// TwinCAT 3 PLC project UlyssesToolBox
// Title: UlyssesToolBox
// Company: NoCompany
// ProjectVersion: 1.0.0.1
// ProgramVersion: 3.1.4024.0
// project tree:
//   TF04Controller/TempController/ EasyTemp.TcPOU, E_EasyTempState.TcDUT, E_TuneMode.TcDUT, FB_TempSimu.TcPOU, ST_EasyTempPara.TcDUT
//   TF05Motion/SimpleAxis/ E_MoveMode.TcDUT, E_SimpleAxisState.TcDUT, FB_SimpleAxis.TcPOU, ST_AxisSettings.TcDUT
//   TF06Connectivity/TCPIP/ FB_TcpSendReceive.TcPOU, FB_TcpSendReceiving.TcPOU, FB_TcpSendReceivingQueue.TcPOU
//   TF06Connectivity/TCPIP/SimpleClient/ SimpleTcpClient.TcPOU, stConnState.TcDUT, stSktPara.TcDUT
//   TF06Connectivity/TCPIP/TcpTaskQueue2/ FB_SimpleTcpTaskQueue2.TcPOU, ST_TcpTask2.TcDUT, ST_TcpTaskBuffer2.TcDUT
//   TF06Connectivity/TCPIP/TcpTaskQueue/ FB_SimpleTcpTaskQueue.TcPOU, ST_TcpTask.TcDUT, ST_TcpTaskBuffer.TcDUT
//   TF06Connectivity/TCPIP/[obsolete]/ FB_TcpSendReceivingHistroy.TcPOU
//   TF11PlcSystem/AnalogScale/ AnalogScale.TcPOU, AnalogScaleWithAlarm.TcPOU
//   TF11PlcSystem/ET_DoubleBuffer/ DataFileLogger.TcPOU, DoubleBuffer.TcPOU, HRESULT_TO_ADSERROR.TcPOU
//   TF11PlcSystem/File/ FB_FileHandler.TcPOU
//   TF11PlcSystem/IO/ DI_Button.TcPOU, DI_Input.TcPOU, Input.TcPOU, Output.TcPOU
//   TF11PlcSystem/Logger/ E_LogFileSplitMode.TcDUT, ULogger.TcPOU
//   TF11PlcSystem/System/File/ FB_File.TcPOU
//   TF11PlcSystem/System/Pendulum4Tc/ Constants.TcPOU, Day.TcPOU, GVLPendulum.TcGVL, Pendulum4Tc.TcPOU, PtDateTime.TcPOU, PtHelper.TcPOU, PtInterval.TcPOU, PtTimeSource.TcPOU
//   TF11PlcSystem/System/Pendulum4Tc/DUTs/ E_TimeSource.TcDUT, PtWeekDay.TcTLEO, ST_WinsowsTimeZone.TcDUT
//   TF11PlcSystem/System/Pendulum4Tc/Functions/ F_TzInfoBiasToTzStr.TcPOU
//   TF11PlcSystem/System/Pendulum4Tc/Helper/ calcDayNumber.TcPOU, calcPreciseDiff.TcPOU, isDateTimeEqual.TcPOU, isLeapYear.TcPOU, PtPreciseDiff.TcPOU
//   TF11PlcSystem/System/Pendulum4Tc/Interface/ I_PtDateTime.TcIO, I_PtInterval.TcIO, I_PtTimesource.TcIO
//   TF11PlcSystem/System/SystemInfo/ System_AppInfo.TcPOU, System_IpcInfo.TcPOU, System_TaskInfo.TcPOU
//   TF11PlcSystem/System/ SystemPulses.TcPOU
//   TF11PlcSystem/System/Time/DataTypes/ ST_TimeConvertor.TcDUT
//   TF11PlcSystem/System/Time/FunctionBlocks/ FB_TimeConvertorM.TcPOU, FB_Time_Task.TcPOU, Pulse.TcPOU, TimeConvertor.TcPOU
//   TF11PlcSystem/System/Time/Functions/ F_FormatTime.TcPOU, F_SYSTEMTIME_TO_String6.TcPOU
//   TF11PlcSystem/System/Time/[obsolete]/ Base_SysTime.TcPOU, FB_TimeConvertor0.TcPOU, F_TimeStamp13_TO_SYSTEMTIME.TcPOU, PulseWrong.TcPOU
// (motion and I/O tree: see PLC project plc851)
// real-time tasks:
//   TASK PlcTask: cycle T#10ms, priority 20, ADS port 350

// ---- TF04Controller/TempController/E_EasyTempState.TcDUT
{attribute 'qualified_only'}
{attribute 'strict'}
TYPE E_EasyTempState :
(
	Stopped := 0,
	Running := 1,
	Tuning := 2,
	Resetting := 99
);
END_TYPE

// ---- TF04Controller/TempController/E_TuneMode.TcDUT
{attribute 'qualified_only'}
{attribute 'strict'}
TYPE E_TuneMode :
(
	Normal := 0,
	Fast := 1,
	Slow :=2
);
END_TYPE

// ---- TF04Controller/TempController/ST_EasyTempPara.TcDUT
TYPE ST_EasyTempPara :
STRUCT
	bTuned : BOOL;
	stPID : ST_CTRL_ParaController;
	stPara: ST_CTRL_TempCtrlParameter;
END_STRUCT
END_TYPE

// ---- TF05Motion/SimpleAxis/E_MoveMode.TcDUT
{attribute 'qualified_only'}
{attribute 'strict'}
TYPE E_MoveMode :
(
	NotMove := 0,
	MoveAbs := 1,
	MoveMod := 2,
	MoveRel := 3

);
END_TYPE

// ---- TF05Motion/SimpleAxis/E_SimpleAxisState.TcDUT
{attribute 'qualified_only'}
{attribute 'strict'}
TYPE E_SimpleAxisState :
(
	Waiting := 0,
	BeforeJog := 10,
	Joging :=11,
	JogDone := 18,
	
	BeforeMovePos :=20,
	MovingAbs := 21,
	MovingMod :=23,
	MovingRel := 24,
	MovePosDone := 28,
	
	BeforeMoveVelo := 30,
	MovingVelo := 31,
	MoveVeloStop := 32,
	MoveVeloDone := 38,
	
	
	BeforeHoming := 50,
	Homing :=51,
	FinishHoming := 52,
	HomeToZero := 53,
	HomeDone :=58,

	Aborted := 90,
	Error :=99

);
END_TYPE

// ---- TF05Motion/SimpleAxis/ST_AxisSettings.TcDUT
TYPE ST_AxisSettings :
STRUCT
	MovePosAcc : LREAL;
	MovePosDec : LREAL;
	MovePosJerk : LREAL;
	
	MoveVeloAcc : LREAL;
	MoveVeloDec : LREAL;
	MoveVeloJerk : LREAL;
	MoveVeloDirection : MC_Direction := MC_Positive_Direction;
	
	JogAcc : LREAL;
	JogDec : LREAL;
	JogJerk : LREAL;
	
	HomeVelo : LREAL := 10;
	HomeAcc : LREAL;
	HomeDec : LREAL;
	HomeJerk : LREAL;
	HomeSetpos : LREAL := 0;
	HomeSignal : BOOL;
	HomePosLimit : BOOL;
	HomeNegLimit : BOOL;
END_STRUCT
END_TYPE

// ---- TF06Connectivity/TCPIP/SimpleClient/stConnState.TcDUT
TYPE stConnState :
STRUCT
	bConnected : BOOL;
	hSocket : T_HSOCKET;
	eState : E_SocketConnectionState;
	bError : BOOL;
	nErrId : UDINT;
END_STRUCT
END_TYPE

// ---- TF06Connectivity/TCPIP/SimpleClient/stSktPara.TcDUT
TYPE stSktPara :
STRUCT
	AutoReconnect : BOOL;
	EnableSendLog : BOOL;
	EnableRecvLog : BOOL;
	SendRecvTimeOut : TIME := T#3S;
	
END_STRUCT
END_TYPE

// ---- TF06Connectivity/TCPIP/TcpTaskQueue2/ST_TcpTask2.TcDUT
{attribute 'pack_mode' := '1'}
TYPE ST_TcpTask2 :
STRUCT
	TaskName : STRING(24);
	TaskType : INT; (* 0:Once, 1:Regular *)
	pData : PVOID;
	nData : UDINT;
END_STRUCT
END_TYPE

// ---- TF06Connectivity/TCPIP/TcpTaskQueue2/ST_TcpTaskBuffer2.TcDUT
{attribute 'pack_mode' := '1'}
TYPE ST_TcpTaskBuffer2 :
STRUCT
	BufferInfo : UDINT;
	TaskData : ST_TcpTask2;
END_STRUCT
END_TYPE

// ---- TF06Connectivity/TCPIP/TcpTaskQueue/ST_TcpTask.TcDUT
{attribute 'pack_mode' := '1'}
TYPE ST_TcpTask :
STRUCT
	TaskName : STRING(24);
	TaskType : INT; (* 0:Once, 1:Regular *)
	TaskData : ARRAY[0..255] OF BYTE;
END_STRUCT
END_TYPE

// ---- TF06Connectivity/TCPIP/TcpTaskQueue/ST_TcpTaskBuffer.TcDUT
{attribute 'pack_mode' := '1'}
TYPE ST_TcpTaskBuffer :
STRUCT
	BufferInfo : ARRAY[0..3] OF BYTE;
	TaskData : ST_TcpTask;
END_STRUCT
END_TYPE

// ---- TF11PlcSystem/Logger/E_LogFileSplitMode.TcDUT
{attribute 'qualified_only'}
{attribute 'strict'}
TYPE E_LogFileSplitMode :
(
	eDontSplit := 0,
	eSplitByDay := 1,
	eSplitByHour := 2
);
END_TYPE

// ---- TF11PlcSystem/System/Pendulum4Tc/DUTs/E_TimeSource.TcDUT
{attribute 'qualified_only'}
{attribute 'strict'}
TYPE E_TimeSource :
(
	FileTime := 0,
	DcTaskInfo := 1,
	fbLocalSystemTime := 2
);
END_TYPE

// ---- TF11PlcSystem/System/Pendulum4Tc/DUTs/PtWeekDay.TcTLEO
{attribute 'qualified_only'}
{attribute 'strict'}
TYPE PtWeekDay :
(
	MONDAY := 0,
    TUESDAY := 1,
    WEDNESDAY := 2,
    THURSDAY := 3,
    FRIDAY := 4,
    SATURDAY := 5,
    SUNDAY := 6
);
END_TYPE

// ---- TF11PlcSystem/System/Pendulum4Tc/DUTs/ST_WinsowsTimeZone.TcDUT
TYPE ST_WinsowsTimeZone :
STRUCT
	AUS_Central_Standard_Time	: STRING	:=	 'Australia/Darwin';
	AUS_Eastern_Standard_Time	: STRING	:=	 'Australia/Sydney';
	Afghanistan_Standard_Time	: STRING	:=	 'Asia/Kabul';
	Alaskan_Standard_Time	: STRING	:=	 'America/Anchorage';
	Aleutian_Standard_Time	: STRING	:=	 'America/Adak';
	Altai_Standard_Time	: STRING	:=	 'Asia/Barnaul';
	Arab_Standard_Time	: STRING	:=	 'Asia/Riyadh';
	Arabian_Standard_Time	: STRING	:=	 'Asia/Dubai';
	Arabic_Standard_Time	: STRING	:=	 'Asia/Baghdad';
	Argentina_Standard_Time	: STRING	:=	 'America/Buenos_Aires';
	Astrakhan_Standard_Time	: STRING	:=	 'Europe/Astrakhan';
	Atlantic_Standard_Time	: STRING	:=	 'America/Halifax';
	Aus_Central_Wdot_Standard_Time	: STRING	:=	 'Australia/Eucla';
	Azerbaijan_Standard_Time	: STRING	:=	 'Asia/Baku';
	Azores_Standard_Time	: STRING	:=	 'Atlantic/Azores';
	Bahia_Standard_Time	: STRING	:=	 'America/Bahia';
	Bangladesh_Standard_Time	: STRING	:=	 'Asia/Dhaka';
	Belarus_Standard_Time	: STRING	:=	 'Europe/Minsk';
	Bougainville_Standard_Time	: STRING	:=	 'Pacific/Bougainville';
	Canada_Central_Standard_Time	: STRING	:=	 'America/Regina';
	Cape_Verde_Standard_Time	: STRING	:=	 'Atlantic/Cape_Verde';
	Caucasus_Standard_Time	: STRING	:=	 'Asia/Yerevan';
	Cendot_Australia_Standard_Time	: STRING	:=	 'Australia/Adelaide';
	Central_America_Standard_Time	: STRING	:=	 'America/Guatemala';
	Central_Asia_Standard_Time	: STRING	:=	 'Asia/Almaty';
	Central_Brazilian_Standard_Time	: STRING	:=	 'America/Cuiaba';
	Central_Europe_Standard_Time	: STRING	:=	 'Europe/Budapest';
	Central_European_Standard_Time	: STRING	:=	 'Europe/Warsaw';
	Central_Pacific_Standard_Time	: STRING	:=	 'Pacific/Guadalcanal';
	Central_Standard_Time	: STRING	:=	 'America/Chicago';
	Central_Standard_Time_Mexico	: STRING	:=	 'America/Mexico_City';
	Chatham_Islands_Standard_Time	: STRING	:=	 'Pacific/Chatham';
	China_Standard_Time	: STRING	:=	 'Asia/Shanghai';
	Cuba_Standard_Time	: STRING	:=	 'America/Havana';
	Dateline_Standard_Time	: STRING	:=	 'Etc/GMT+12';
	Edot_Africa_Standard_Time	: STRING	:=	 'Africa/Nairobi';
	Edot_Australia_Standard_Time	: STRING	:=	 'Australia/Brisbane';
	Edot_Europe_Standard_Time	: STRING	:=	 'Europe/Chisinau';
	Edot_South_America_Standard_Time	: STRING	:=	 'America/Sao_Paulo';
	Easter_Island_Standard_Time	: STRING	:=	 'Pacific/Easter';
	Eastern_Standard_Time	: STRING	:=	 'America/New_York';
	Eastern_Standard_Time_Mexico	: STRING	:=	 'America/Cancun';
	Egypt_Standard_Time	: STRING	:=	 'Africa/Cairo';
	Ekaterinburg_Standard_Time	: STRING	:=	 'Asia/Yekaterinburg';
	FLE_Standard_Time	: STRING	:=	 'Europe/Kiev';
	Fiji_Standard_Time	: STRING	:=	 'Pacific/Fiji';
	GMT_Standard_Time	: STRING	:=	 'Europe/London';
	GTB_Standard_Time	: STRING	:=	 'Europe/Bucharest';
	Georgian_Standard_Time	: STRING	:=	 'Asia/Tbilisi';
	Greenland_Standard_Time	: STRING	:=	 'America/Godthab';
	Greenwich_Standard_Time	: STRING	:=	 'Atlantic/Reykjavik';
	Haiti_Standard_Time	: STRING	:=	 'America/Port-au-Prince';
	Hawaiian_Standard_Time	: STRING	:=	 'Pacific/Honolulu';
	India_Standard_Time	: STRING	:=	 'Asia/Calcutta';
	Iran_Standard_Time	: STRING	:=	 'Asia/Tehran';
	Israel_Standard_Time	: STRING	:=	 'Asia/Jerusalem';
	Jordan_Standard_Time	: STRING	:=	 'Asia/Amman';
	Kaliningrad_Standard_Time	: STRING	:=	 'Europe/Kaliningrad';
	Korea_Standard_Time	: STRING	:=	 'Asia/Seoul';
	Libya_Standard_Time	: STRING	:=	 'Africa/Tripoli';
	Line_Islands_Standard_Time	: STRING	:=	 'Pacific/Kiritimati';
	Lord_Howe_Standard_Time	: STRING	:=	 'Australia/Lord_Howe';
	Magadan_Standard_Time	: STRING	:=	 'Asia/Magadan';
	Magallanes_Standard_Time	: STRING	:=	 'America/Punta_Arenas';
	Marquesas_Standard_Time	: STRING	:=	 'Pacific/Marquesas';
	Mauritius_Standard_Time	: STRING	:=	 'Indian/Mauritius';
	Middle_East_Standard_Time	: STRING	:=	 'Asia/Beirut';
	Montevideo_Standard_Time	: STRING	:=	 'America/Montevideo';
	Morocco_Standard_Time	: STRING	:=	 'Africa/Casablanca';
	Mountain_Standard_Time	: STRING	:=	 'America/Denver';
	Mountain_Standard_Time_Mexico	: STRING	:=	 'America/Chihuahua';
	Myanmar_Standard_Time	: STRING	:=	 'Asia/Rangoon';
	Ndot_Central_Asia_Standard_Time	: STRING	:=	 'Asia/Novosibirsk';
	Namibia_Standard_Time	: STRING	:=	 'Africa/Windhoek';
	Nepal_Standard_Time	: STRING	:=	 'Asia/Katmandu';
	New_Zealand_Standard_Time	: STRING	:=	 'Pacific/Auckland';
	Newfoundland_Standard_Time	: STRING	:=	 'America/St_Johns';
	Norfolk_Standard_Time	: STRING	:=	 'Pacific/Norfolk';
	North_Asia_East_Standard_Time	: STRING	:=	 'Asia/Irkutsk';
	North_Asia_Standard_Time	: STRING	:=	 'Asia/Krasnoyarsk';
	North_Korea_Standard_Time	: STRING	:=	 'Asia/Pyongyang';
	Omsk_Standard_Time	: STRING	:=	 'Asia/Omsk';
	Pacific_SA_Standard_Time	: STRING	:=	 'America/Santiago';
	Pacific_Standard_Time	: STRING	:=	 'America/Los_Angeles';
	Pacific_Standard_Time_Mexico	: STRING	:=	 'America/Tijuana';
	Pakistan_Standard_Time	: STRING	:=	 'Asia/Karachi';
	Paraguay_Standard_Time	: STRING	:=	 'America/Asuncion';
	Romance_Standard_Time	: STRING	:=	 'Europe/Paris';
	Russia_Time_Zone_10	: STRING	:=	 'Asia/Srednekolymsk';
	Russia_Time_Zone_11	: STRING	:=	 'Asia/Kamchatka';
	Russia_Time_Zone_3	: STRING	:=	 'Europe/Samara';
	Russian_Standard_Time	: STRING	:=	 'Europe/Moscow';
	SA_Eastern_Standard_Time	: STRING	:=	 'America/Cayenne';
	SA_Pacific_Standard_Time	: STRING	:=	 'America/Bogota';
	SA_Western_Standard_Time	: STRING	:=	 'America/La_Paz';
	SE_Asia_Standard_Time	: STRING	:=	 'Asia/Bangkok';
	Saint_Pierre_Standard_Time	: STRING	:=	 'America/Miquelon';
	Sakhalin_Standard_Time	: STRING	:=	 'Asia/Sakhalin';
	Samoa_Standard_Time	: STRING	:=	 'Pacific/Apia';
	Sao_Tome_Standard_Time	: STRING	:=	 'Africa/Sao_Tome';
	Saratov_Standard_Time	: STRING	:=	 'Europe/Saratov';
	Singapore_Standard_Time	: STRING	:=	 'Asia/Singapore';
	South_Africa_Standard_Time	: STRING	:=	 'Africa/Johannesburg';
	Sri_Lanka_Standard_Time	: STRING	:=	 'Asia/Colombo';
	Sudan_Standard_Time	: STRING	:=	 'Africa/Khartoum';
	Syria_Standard_Time	: STRING	:=	 'Asia/Damascus';
	Taipei_Standard_Time	: STRING	:=	 'Asia/Taipei';
	Tasmania_Standard_Time	: STRING	:=	 'Australia/Hobart';
	Tocantins_Standard_Time	: STRING	:=	 'America/Araguaina';
	Tokyo_Standard_Time	: STRING	:=	 'Asia/Tokyo';
	Tomsk_Standard_Time	: STRING	:=	 'Asia/Tomsk';
	Tonga_Standard_Time	: STRING	:=	 'Pacific/Tongatapu';
	Transbaikal_Standard_Time	: STRING	:=	 'Asia/Chita';
	Turkey_Standard_Time	: STRING	:=	 'Europe/Istanbul';
	Turks_And_Caicos_Standard_Time	: STRING	:=	 'America/Grand_Turk';
	US_Eastern_Standard_Time	: STRING	:=	 'America/Indianapolis';
	US_Mountain_Standard_Time	: STRING	:=	 'America/Phoenix';
	UTC	: STRING	:=	 'Etc/GMT';
	UTCplus12	: STRING	:=	 'Etc/GMT-12';
	UTCplus13	: STRING	:=	 'Etc/GMT-13';
	UTCminus02	: STRING	:=	 'Etc/GMT+2';
	UTCminus08	: STRING	:=	 'Etc/GMT+8';
	UTCminus09	: STRING	:=	 'Etc/GMT+9';
	UTCminus11	: STRING	:=	 'Etc/GMT+11';
	Ulaanbaatar_Standard_Time	: STRING	:=	 'Asia/Ulaanbaatar';
	Venezuela_Standard_Time	: STRING	:=	 'America/Caracas';
	Vladivostok_Standard_Time	: STRING	:=	 'Asia/Vladivostok';
	Wdot_Australia_Standard_Time	: STRING	:=	 'Australia/Perth';
	Wdot_Central_Africa_Standard_Time	: STRING	:=	 'Africa/Lagos';
	Wdot_Europe_Standard_Time	: STRING	:=	 'Europe/Berlin';
	Wdot_Mongolia_Standard_Time	: STRING	:=	 'Asia/Hovd';
	West_Asia_Standard_Time	: STRING	:=	 'Asia/Tashkent';
	West_Bank_Standard_Time	: STRING	:=	 'Asia/Hebron';
	West_Pacific_Standard_Time	: STRING	:=	 'Pacific/Port_Moresby';
	Yakutsk_Standard_Time	: STRING	:=	 'Asia/Yakutsk';

END_STRUCT
END_TYPE

// ---- TF11PlcSystem/System/Time/DataTypes/ST_TimeConvertor.TcDUT
TYPE ST_TimeConvertor :
STRUCT
		(* #########################  System  ######################### *)
		
	(* Alias: -- *)
	(* Size: 32-bit *)
	(* Range: 0=>1970-01-01 2^32-1=>2106-02-07 *)
	(* Resolution: 1s, only the day is displayed *)
	(* https://infosys.beckhoff.com/english.php?content=../content/1033/tc3_plc_intro/2529415819.html&id=7132877304198979715 *)
	(* Native *)
	Date_D : DATE;
	
	(* Alias: -- *)
	(* Size: 32-bit *)
	(* Range: 0=>00:00:00.000 86399999=>23:59:59.999 *)
	(* Resolution: 1ms *)
	(* https://infosys.beckhoff.com/english.php?content=../content/1033/tc3_plc_intro/2529415819.html&id=7132877304198979715 *)
	(* Native *)
	TimeOfDay_TOD : TIME_OF_DAY;
	
	(* Alias: -- *)
	(* Size: 32-bit *)
	(* Range: 0=>1970-01-01 00:00:00 2^32-1=>2106-02-07 06:28:15 *)
	(* Resolution: 1s *)
	(* https://infosys.beckhoff.com/english.php?content=../content/1033/tc3_plc_intro/2529415819.html&id=7132877304198979715 *)
	(* Native *)
	DateAndTime_DT : DATE_AND_TIME;
	
	(* Alias: -- *)
	(* Size: 64-bit *)
	(* Range: 0=>1970-01-01 2^64-1=>2554-07-21 *)
	(* Resolution: 1ns *)
	(* https://infosys.beckhoff.com/english.php?content=../content/1033/tc3_plc_intro/2529415819.html&id=7132877304198979715 *)
	(* Only For >=4026.0 *)
	//LDate_LDT : LDATE;
	
	(* Alias: -- *)
	(* Size: 64-bit *)
	(* Range: 0=>00:00:00.000000000 2^64-1=>23:59:59.999999999 *)
	(* Resolution: 1ns *)
	(* https://infosys.beckhoff.com/english.php?content=../content/1033/tc3_plc_intro/2529415819.html&id=7132877304198979715 *)
	(* Only For >=4026.0 *)
	//LTimeOfDay_LTOD : LTIME_OF_DAY;
	
	(* Alias: -- *)
	(* Size: 64-bit *)
	(* Range: 0=>1970-01-01 00:00:00.000000000 2^64-1=>2554-07-21 23:34:33.709551615 *)
	(* Resolution: 1ns *)
	(* https://infosys.beckhoff.com/english.php?content=../content/1033/tc3_plc_intro/2529415819.html&id=7132877304198979715 *)
	(* Only For >=4026.0 *)
	//LDateAndTime_LDT : LDATE_AND_TIME;
	
		(* #########################  Tc2_Utilities  ######################### *)
	
	(* Alias: T_ULARGE_INTEGER -> Struct of 2 DWORD *)
	(* Size: 64-bit *)
	(* Range: -- *)
	(* Resolution: 100ns *)
	(* obsolete! *)
	FileTime : T_FILETIME;
	
	(* Alias: ULINT *)
	(* Size: 64-bit *)
	(* Range: 0=>1601-01-01 00:00:00.0000000 2^64-1=>2185-11-09 23:34:33.9999999 *)
	(* Resolution: 100ns *)
	(* https://infosys.beckhoff.com/english.php?content=../content/1033/tcplclib_tc2_utilities/10462547339.html&id= *)
	(* Recommend! *)
	FileTime64 : T_FILETIME64;
	
	(* Alias: Struct of 8 WORD *)
	(* Size: 128-bit *)
	(* Range: 1970-01-01 Sunday 00:00:00.000  2106-12-31 Saturday 23:59:59.999 *)
	(* Resolution: 1ms *)
	(* https://infosys.beckhoff.com/english.php?content=../content/1033/tcplclib_tc2_utilities/35393035.html&id=8702657298802174446 *)
	(* Recommend! *)
	TimeStruct : TIMESTRUCT;
	
	(* Alias: Struct of 6 WORD *)
	(* Size: 96-bit *)
	(* Range: Week0 Day0 00:00:00.000  Week65535 Day7 23:59:59.999 *)
	(* Resolution: 1ms *)
	(* https://infosys.beckhoff.com/english.php?content=../content/1033/tcplclib_tc2_utilities/35353099.html&id=8265378500365774535 *)
	(* What's this??  weeks + days *)
	(* NOT Recommend! *)
	OtStruct : OTSTRUCT;
	
		(* #########################  Tc2_EtherCAT  ######################### *)
		
	(* Alias: T_ULARGE_INTEGER -> Struct of 2 DWORD *)
	(* Size: 64-bit *)
	(* Range: -- *)
	(* Resolution: 1ns *)
	(* obsolete! *)
	DcTime : T_DCTIME;
	
	(* Alias: UDINT *)
	(* Size: 32-bit *)
	(* Range: +-2147s *)
	(* Resolution: 1ns *)
	(* NOT Recommend! *)
	DcTime32 : T_DCTIME32; 
	
	(* Alias: ULINT *)
	(* Size: 64-bit *)
	(* Range: 0=>2000-01-01 00:00:00.000000000 2^64-1=>2584-11-09 23:34:33.999999999 *)
	(* Resolution: 1ns *)
	(* Recommend! *)
	DcTime64 : T_DCTIME64;

		(* #########################  Custom & Others  ######################### *)
	
	Unix : UDINT;
	UnixEx : ULINT;
	//Unix64
END_STRUCT
END_TYPE

// ---- TF11PlcSystem/System/Pendulum4Tc/GVLPendulum.TcGVL
//{attribute 'qualified_only'}
VAR_GLOBAL
	Pendulum : Pendulum4Tc;
END_VAR

// ---- TF11PlcSystem/System/Pendulum4Tc/Interface/I_PtDateTime.TcIO
INTERFACE I_PtDateTime

END_INTERFACE

// ---- TF11PlcSystem/System/Pendulum4Tc/Interface/I_PtInterval.TcIO
INTERFACE I_PtInterval

METHOD inMonth : DINT
VAR_INPUT
END_VAR
END_METHOD

METHOD inYears : DINT
VAR_INPUT
END_VAR
END_METHOD

END_INTERFACE

// ---- TF11PlcSystem/System/Pendulum4Tc/Interface/I_PtTimesource.TcIO
INTERFACE I_PtTimesource

METHOD getDateTime : PtDateTime
VAR_INPUT
END_VAR
END_METHOD

END_INTERFACE

// ---- TF11PlcSystem/System/Pendulum4Tc/Pendulum4Tc.TcPOU
FUNCTION_BLOCK Pendulum4Tc
VAR_INPUT
	TimeSourceDateTime : I_PtTimesource;
END_VAR
VAR_OUTPUT
END_VAR
VAR
	_DateTime : PtDateTime;
	_Interval : PtInterval;
END_VAR


_DateTime := TimeSourceDateTime.getDateTime();

METHOD New : PtDateTime
VAR_INPUT
	Year : DINT;
	Month : DINT;
	Day : DINT;
	Hour : DINT;
	Minute : DINT;
	Second : DINT;
	Microsecond : DINT;
	TimeZone : DINT;
END_VAR
New.Set(
	Year:= Year, 
	Month:= Month, 
	Day:= Day, 
	Hour:= Hour, 
	Minute:= Minute, 
	Second:= Second, 
	Microsecond:= Microsecond, 
	TimeZone:= TimeZone);
END_METHOD

METHOD Now : PtDateTime
VAR_INPUT
END_VAR
Now := _DateTime;
END_METHOD

END_FUNCTION_BLOCK

// ---- TF11PlcSystem/System/Pendulum4Tc/PtDateTime.TcPOU
FUNCTION_BLOCK PtDateTime IMPLEMENTS I_PtDateTime
VAR_INPUT
END_VAR
VAR_OUTPUT
END_VAR
VAR
	_Year : DINT;
	_Month : DINT;
	_Day : DINT;
	_Hour : DINT;
	_Minute : DINT;
	_Second : DINT;
	_Microsecond : DINT;
	_TimeZone : DINT;
	
END_VAR

PROPERTY Day : DINT
GET
Day := _Day;
END_GET
SET
_Day := Day;
END_SET
END_PROPERTY

METHOD Diff : I_PtInterval
VAR_INPUT
	TargetDateTime : PtDateTime;
END_VAR
//Diff.Set(THIS^,TargetDateTime,TRUE);
Pendulum._interval.Set(THIS^,TargetDateTime,TRUE);
Diff := Pendulum._interval;
END_METHOD

PROPERTY Hour : DINT
GET
Hour := _Hour;
END_GET
SET
_Hour := Hour;
END_SET
END_PROPERTY

PROPERTY Microsecond : DINT
GET
Microsecond := _Microsecond;
END_GET
SET
_Microsecond := Microsecond;
END_SET
END_PROPERTY

PROPERTY Minute : DINT
GET
Minute := _Minute;
END_GET
SET
_Minute := Minute;
END_SET
END_PROPERTY

PROPERTY Month : DINT
GET
Month := _Month;
END_GET
SET
_Month := Month;
END_SET
END_PROPERTY

PROPERTY Second : DINT
GET
Second := _Second;
END_GET
SET
_Second := Second;
END_SET
END_PROPERTY

METHOD Set //: PtDateTime
VAR_INPUT
	Year : DINT;
	Month : DINT;
	Day : DINT;
	Hour : DINT;
	Minute : DINT;
	Second : DINT;
	Microsecond : DINT;
	TimeZone : DINT;
END_VAR
THIS^._Year := Year;
THIS^._Month := Month;
THIS^._Day := Day;
THIS^._Hour := Hour;
THIS^._Minute := Minute;
THIS^._Second := Second;
THIS^._Microsecond := Microsecond;
THIS^._TimeZone := TimeZone;
END_METHOD

PROPERTY TimeZone : DINT
GET
TimeZone := _TimeZone;
END_GET
SET
_TimeZone := TimeZone;
END_SET
END_PROPERTY

PROPERTY Year : DINT
GET
Year := _Year;
END_GET
SET
_Year := Year;
END_SET
END_PROPERTY

END_FUNCTION_BLOCK

// ---- TF11PlcSystem/System/Pendulum4Tc/Day.TcPOU
FUNCTION_BLOCK Day
VAR_INPUT
	
END_VAR
VAR_OUTPUT
END_VAR
VAR
END_VAR

END_FUNCTION_BLOCK

// ---- TF11PlcSystem/System/Pendulum4Tc/PtInterval.TcPOU
FUNCTION_BLOCK PtInterval IMPLEMENTS I_PtInterval
VAR_INPUT
END_VAR
VAR_OUTPUT
END_VAR
VAR
	_Start : PtDateTime;
	_End : PtDateTime;
	_Absolute : BOOL;
	
	_DeltaYears : DINT;
	_DeltaMonths : DINT;
	_DeltaDays : DINT;
END_VAR

PROPERTY Absolute : BOOL
GET
Absolute := _Absolute;
END_GET
SET
_Absolute := Absolute;
END_SET
END_PROPERTY

PROPERTY End : PtDateTime
GET
End := _End;
END_GET
SET
_End := End;
END_SET
END_PROPERTY

METHOD inMonth : DINT
VAR_INPUT
END_VAR
inMonth := ABS(_Start.Month - _End.Month);
END_METHOD

METHOD inYears : DINT
VAR_INPUT
END_VAR
inYears := ABS(_Start.Year - _End.Year);
END_METHOD

METHOD Set //: BOOL
VAR_INPUT
	Start : PtDateTime;
	End : PtDateTime;
	Absolute : BOOL;
END_VAR
_Start := Start;
_End := End;
_Absolute := Absolute;

_DeltaYears := ABS(_Start.Year - _End.Year);
_DeltaMonths := ABS(_Start.Month - _End.Month);
_DeltaDays := ABS(_Start.Day - End.Day);
END_METHOD

PROPERTY Start : PtDateTime
GET
END_GET
SET
_Start := Start;
END_SET
END_PROPERTY

END_FUNCTION_BLOCK

// ---- TF04Controller/TempController/EasyTemp.TcPOU
FUNCTION_BLOCK EasyTemp
VAR_INPUT
	bStart : BOOL;
	bTune : BOOL;
	TuneMode : E_TuneMode := E_TuneMode.Normal;
	bReset : BOOL;
	SensorTemp : LREAL;
	TargetTemp : LREAL;
	
END_VAR
VAR_IN_OUT
	EasyTempPara : ST_EasyTempPara;
END_VAR
VAR_OUTPUT
	State : E_EasyTempState;
	fAnalog : LREAL;
	bPWMPos : BOOL;
	bPWMNeg : BOOL;
	bDigPos : BOOL;
	bDigNeg : BOOL;
	fMaxOverShoot: LREAL;
	tStartUpTime: TIME;
	eControlState: Tc2_TempController.E_CTRL_STATE;
	bError: BOOL;
	eErrorId: Tc2_TempController.E_CTRL_ErrorCodes;
	fTempVelo: LREAL;
	
END_VAR
VAR

	rTrigStart : R_TRIG;
	fTrigStart : F_TRIG;
	rTrigTune : R_TRIG;
	rTrigReset : R_TRIG;
	//状态机
	_State : E_EasyTempState;
	rTrigStateReq : R_TRIG;
	fbTemp : FB_CTRL_TempController;


END_VAR

ParaUpdate();


rTrigStart(CLK:= bStart, Q=> );
fTrigStart(CLK:= bStart, Q=> );
rTrigTune(CLK:= bTune, Q=> );
rTrigStateReq(CLK:= rTrigStart.Q XOR fTrigStart.Q XOR rTrigTune.Q, Q=> );
rTrigReset(CLK:= bReset, Q=> );
IF rTrigReset.Q THEN
	_State := E_EasyTempState.Resetting;
END_IF
CASE _State OF
E_EasyTempState.Stopped:
	IF rTrigStateReq.Q THEN
		IF rTrigStart.Q THEN
			IF EasyTempPara.bTuned THEN
				_State := E_EasyTempState.Running;
			END_IF
		ELSIF fTrigStart.Q THEN
			//no action
		ELSIF rTrigTune.Q THEN
			_State := E_EasyTempState.Tuning;
		END_IF
	END_IF
	fbTemp.eCtrlMode := E_CTRL_MODE.eCTRL_MODE_IDLE;
	
E_EasyTempState.Tuning:
	IF rTrigStateReq.Q THEN
		IF rTrigStart.Q THEN
			//no action
		ELSIF fTrigStart.Q THEN
			//no action
		ELSIF rTrigTune.Q THEN
			//no action
		END_IF
	END_IF
	IF fbTemp.eCtrlMode = E_CTRL_MODE.eCTRL_MODE_TUNE AND
		(fbTemp.eCtrlState = E_CTRL_STATE.eCTRL_STATE_TUNED OR fbTemp.bError)THEN
		_State := E_EasyTempState.Stopped;
		IF fbTemp.eCtrlState = E_CTRL_STATE.eCTRL_STATE_TUNED THEN
			EasyTempPara.stPID := fbTemp.sParaControllerInternal;
			EasyTempPara.bTuned := TRUE;
		END_IF
	ELSE
		fbTemp.eCtrlMode := E_CTRL_MODE.eCTRL_MODE_TUNE;
	END_IF
	
E_EasyTempState.Running:
	IF rTrigStateReq.Q THEN
		IF rTrigStart.Q THEN
			//no action
		ELSIF fTrigStart.Q THEN
			_State := E_EasyTempState.Stopped;
		ELSIF rTrigTune.Q THEN
			//no action
		END_IF
	END_IF
	fbTemp.eCtrlMode := E_CTRL_MODE.eCTRL_MODE_ACTIVE;
E_EasyTempState.Resetting:
	fbTemp.eCtrlMode := E_CTRL_MODE.eCTRL_MODE_RESET;
	IF fbTemp.eCtrlState = E_CTRL_STATE.eCTRL_STATE_IDLE THEN
		_State := E_EasyTempState.Stopped;
	END_IF
END_CASE
State := _State;



fbTemp.sParaControllerExternal := EasyTempPara.stPID;
fbTemp.fW1 := TargetTemp;
fbTemp.fX := SensorTemp;
fbTemp(
	eCtrlMode:= , 
	bSelSetpoint:= , 
	fW1:= , 
	fW2:= , 
	fX:= , 
	fYManual:= , 
	bOpenThermocouple:= , 
	bReverseThermocouple:= , 
	bBackVoltage:= , 
	bLeakage:= , 
	bShortCircuit:= , 
	bOpenCircuit:= , 
	sParaControllerExternal:= , 
	sControllerParameter:= EasyTempPara.stPara, 
	fYAnalog=> fAnalog, 
	bYPWMPos=> bPWMPos, 
	bYPWMNeg=> bPWMNeg, 
	bYDigPos=> bDigPos, 
	bYDigNeg=> bDigNeg, 
	dwAlarm=> , 
	fMaxOverShoot=> fMaxOverShoot, 
	tStartUpTime=> tStartUpTime, 
	eCtrlState=> eControlState, 
	sParaControllerInternal=> , 
	bError=> bError, 
	eErrorId=> eErrorId, 
	fYP=> , 
	fYI=> , 
	fYD=> , 
	fTempVelo=> fTempVelo);

METHOD PRIVATE ParaUpdate : BOOL
VAR_INPUT
END_VAR

			(*	常规参数General parameters	*)
(* 控制器操作模式(见下方) *)
(*
eCTRL_ControlMode_HEATING = 1 : 加热
eCTRL_ControlMode_COOLING = 2 : 降温
eCTRL_ControlMode_HEATING_COOLING = 3 : 加热&降温
*)
EasyTempPara.stPara.iMode							:= E_CTRL_ControlMode.eCTRL_ControlMode_HEATING ;
(* 定义发生错误后的行为 *)
(*
eCTRL_ReactionOnFailure_NoFailure : 没有错误
eCTRL_ReactionOnFailure_StopController : 停止
eCTRL_ReactionOnFailure_SetManMode : 设定为手动模式输出
eCTRL_ReactionOnFailure_SetYMax : 设定为最大输出
eCTRL_ReactionOnFailure_SetYMin : 设定为最小输出
eCTRL_ReactionOnFailure_SetYMean : 设定为平均输出
*)
EasyTempPara.stPara.iReactionOnFailure				:= E_CTRL_ReactionOnFailure.eCTRL_ReactionOnFailure_StopController ;
(* TRUE = 外部参数，FALSE = 内部参数 (取决于自整定) *)
EasyTempPara.stPara.bSelCtrlParameterSet			:= TRUE;
(* 报警掩码（见下文）。 *)
(*
Bit0 : 硬件:温度传感器开路,对应bOpenThermocouple引脚
Bit1 : 硬件:温度传感器反接,对应bReverseThermocouple引脚
Bit2 : 硬件:温度传感器电压过高,对应bBackVoltage引脚
Bit4 : 硬件:温度传感器漏电流,对应bLeakage引脚
Bit5 : 硬件:温度传感器短路,对应bShortCircuit引脚
Bit6 : 硬件:温度传感器开路,对应bOpenCircuit引脚
Bit8 : 软件:温度低于L
Bit9 : 软件:温度低于LL
Bit10: 软件:温度高于H
Bit11: 软件:温度高于HH
Bit12: 软件:温度高于AbsoluteHigh
Bit13: 软件:温度低于AbsoluteLow
*)
EasyTempPara.stPara.dwAlarmSupp						:= 16#FF_FF_FF_FF ;
(* 控制器的采样时间。在采样时间的过程中，控制器重新计算控制值。 *)
EasyTempPara.stPara.tCtrlCycleTime					:= T#100MS	 ;
(* 任务周期时间。用这个时间间隔调用FB。 *)
EasyTempPara.stPara.tTaskCycleTime					:= T#10MS ;

			(*	自整定参数Tuning parameters	*)
(* 确定自整定顺序（见下文）。 *)
EasyTempPara.stPara.iTuningMode						:= eCTRL_TuneMode_heating ;
(* 等待时间，直到稳定后再进行自整定。 *)
EasyTempPara.stPara.tTuneStabilisation				:= T#10S;
(* 设定点的百分比值，从该值开始系统切换到闭环控制。 *)
EasyTempPara.stPara.fEndTunePercentHeating			:= 100.0 ;
(* 自整定过程中控制值的阶跃变化。 *)
EasyTempPara.stPara.fYTuneHeating					:= 60.0 ;
(* 加热时切换到自整定时的控制值 *)
EasyTempPara.stPara.fYStableHeating					:= 0 ;
(* 设定点的百分比值，从该值开始系统切换到闭环控制。 *)
EasyTempPara.stPara.fEndTunePercentCooling			:= 20 ;
(* 自整定过程中控制值的阶跃变化。 *)
EasyTempPara.stPara.fYTuneCooling;
(* 冷却时切换到自整定时的控制值 *)
EasyTempPara.stPara.fYStableCooling;
(* 如果不对冷却进行调整，参数切换的比例系数。 *)
EasyTempPara.stPara.fScalingFactor;

			(*	设定值参数Setpoint parameters	*)
(* 最小设定值 *)
EasyTempPara.stPara.fWMin							:=	 15 ;
(* 最大设定值 *)
EasyTempPara.stPara.fWMax							:=	 120 ;
(* FALSE = 无软启动，TRUE = 软启动 *)
EasyTempPara.stPara.bEnableSoftStart;
(* FALSE = 没有斜坡，TRUE = 斜坡。 *)
EasyTempPara.stPara.bEnableRamping;
(* 启动时的设定值 *)
EasyTempPara.stPara.fWStartUp							 ;
(* 与fWStartUp设定点的时间 *)
EasyTempPara.stPara.tStartUp						:= T#10S ;
(* 在启动阶段打开斜坡。 *)
EasyTempPara.stPara.bStartUpRamping					 ;
(* 启动阶段的上升率（斜率）。 *)
EasyTempPara.stPara.fWStartUpVeloPos				:= 0.08 ;
(* 启动阶段的下降率（斜率）。 *)
EasyTempPara.stPara.fWStartUpVeloNeg				:= 0.08 ;
(* 上升率（坡道） *)
EasyTempPara.stPara.fWVeloPos						:= 1 ;
(* 下降率（坡道 *)
EasyTempPara.stPara.fWVeloNeg						:= 1 ;

			(*	实际值参数Actual value parameters	*)
(* 如果为 "true"，实际值过滤器被激活。 *)
EasyTempPara.stPara.bFilter							:= FALSE ;
(* 实际值滤波器的时间常数（一阶P-T1滤波器） *)
EasyTempPara.stPara.tFilter							:= T#100MS ;

			(*	死区参数Deadband parameters	*)
(* TRUE=死区开启，FALSE=死区关闭 *)
EasyTempPara.stPara.bDeadband						:= FALSE ;
(* 死区，单位：度 *)
EasyTempPara.stPara.fEDeadband						:= 1.0 ;
(* TRUE=默认输入死区，FALSE=输出死区，这个不知道什么用，新版本添加的，不用管*)
EasyTempPara.stPara.bDeadbandOnInput;

			(*	控制值参数Control value parameters	*)
(* 过冲最小化器参数，新版本添加的，不知道啥用 *)
EasyTempPara.stPara.bMinimizeOvershoot;
(* 最小化器的控制误差 *)
EasyTempPara.stPara.fEDelta;
(* 过冲最小化器控制值 *)
EasyTempPara.stPara.fYMinimizeOvershoot;
(* 控制值的最小值 *)
EasyTempPara.stPara.fYMin							:= 0 ;
(* 控制值的最大值 *)
EasyTempPara.stPara.fYMax							:= 100 ;
(* 手动操作中的控制值 *)
EasyTempPara.stPara.fYManual						:= 20 ;
(* 出错时的控制值（可设置参数） *)
EasyTempPara.stPara.fYOnFailure;
(* 冷却PWM指定参数 *)
EasyTempPara.stPara.bPWMCool;
(* PWM信号的周期时间 *)
EasyTempPara.stPara.tPWMCycleTime					:= T#100MS ;
(* PWM：最小关闭时间 *)
EasyTempPara.stPara.tPWMMinOffTime;
(* PWM：最小开启时间 *)
EasyTempPara.stPara.tPWMMinOnTime;
(* PWM：从加热到冷却切换时的等待时间 *)
EasyTempPara.stPara.tPWMWaitingTime;
(* PWM信号的周期时间 *)
EasyTempPara.stPara.tPWMCycleTimeCool;
(* PWM：最小关闭时间 *)
EasyTempPara.stPara.tPWMMinOffTimeCool;
(* PWM：最小开启时间 *)
EasyTempPara.stPara.tPWMMinOnTimeCool;
(* PWM：从加热到冷却切换时的等待时间 *)
EasyTempPara.stPara.tPWMWaitingTimeCool;
(* 3点： 关闭阈值 *)
EasyTempPara.stPara.fYThresholdOff;
(* 3点： 开启阈值 *)
EasyTempPara.stPara.fYThresholdOn;
(* 从一个参数集过渡到另一个参数集的周期数 *)
EasyTempPara.stPara.nCyclesForSwitchOver;

			(*	控制器参数Controller parameters	*)
(* 将预控器打开。 *)
EasyTempPara.stPara.bEnablePreController			:= FALSE ;
(* 将开环特性打开，直到接近设定值。 *)
EasyTempPara.stPara.bEnableZones					:= FALSE ;
(* 闭环控制启动时最小值低于设定值的控制误差 *)
EasyTempPara.stPara.fEnableZoneClosedLoopZone;
(* 在主控制器之后打开控制值过滤器。 *)
EasyTempPara.stPara.bEnableCVFilter					:= FALSE ;
(* 选择主控制器之后的控制值过滤器的类型（见下文）。 *)
EasyTempPara.stPara.iFilterType						:= E_CTRL_FilterType.eCTRL_FilterType_AVERAGE ;
(* 选择一种控制算法（见下文）。 *)
EasyTempPara.stPara.iControllerType					:= E_CTRL_ControllerType.eCTRL_ControllerType_PID ;

			(*	报警参数Alarming parameters	*)
(* 切换到备用参数集--尚不支持 *)
EasyTempPara.stPara.bAlternateParameter;
(* 备用参数集的数量--尚未支持 *)
EasyTempPara.stPara.nAlternateParameterSet;
(* 新版本内容，暂时不用管 *)
EasyTempPara.stPara.bPPartInFeedbackPath;
(* 新版本内容，暂时不用管 *)
EasyTempPara.stPara.bDPartInFeedbackPath;
(* L *)
EasyTempPara.stPara.TempLow							:= 80 ;
(* LL *)
EasyTempPara.stPara.TempLowLow						:= 90 ;
(* H *)
EasyTempPara.stPara.TempHigh						:= 110 ;
(* HH *)
EasyTempPara.stPara.TempHighHigh					:= 120 ;
(* 绝对温度上限 *)
EasyTempPara.stPara.TempAbsoluteHigh				:= 150 ;
(* 绝对温度下限 *)
EasyTempPara.stPara.TempAbsoluteLow					:= 50 ;

			(*	进阶参数Expert parameters	*)
CASE TuneMode OF
E_TuneMode.Fast:
	(* PID控制器的微调参数（仅适用于高级用户）。 *)
	EasyTempPara.stPara.fTuneKp							:= 1.2 ;
	(* PID控制器的微调参数（仅适用于高级用户）。 *)
	EasyTempPara.stPara.fTuneTn							:= 2.0 ;
	(* PID控制器的微调参数（仅适用于高级用户）。 *)
	EasyTempPara.stPara.fTuneTv							:= 0.42 ;
	(* PID控制器的微调参数（仅适用于高级用户）。 *)
	EasyTempPara.stPara.fTuneTd							:= 0.25 ;
	
E_TuneMode.Normal:
	(* PID控制器的微调参数（仅适用于高级用户）。 *)
	EasyTempPara.stPara.fTuneKp							:= 1.0 ;
	(* PID控制器的微调参数（仅适用于高级用户）。 *)
	EasyTempPara.stPara.fTuneTn							:= 2.5 ;
	(* PID控制器的微调参数（仅适用于高级用户）。 *)
	EasyTempPara.stPara.fTuneTv							:= 0.42 ;
	(* PID控制器的微调参数（仅适用于高级用户）。 *)
	EasyTempPara.stPara.fTuneTd							:= 0.25 ;
	
E_TuneMode.Slow:
	(* PID控制器的微调参数（仅适用于高级用户）。 *)
	EasyTempPara.stPara.fTuneKp							:= 0.5 ;
	(* PID控制器的微调参数（仅适用于高级用户）。 *)
	EasyTempPara.stPara.fTuneTn							:= 3.0 ;
	(* PID控制器的微调参数（仅适用于高级用户）。 *)
	EasyTempPara.stPara.fTuneTv							:= 1 ;
	(* PID控制器的微调参数（仅适用于高级用户）。 *)
	EasyTempPara.stPara.fTuneTd							:= 0.25 ;

END_CASE
END_METHOD

END_FUNCTION_BLOCK

// ---- TF04Controller/TempController/FB_TempSimu.TcPOU
FUNCTION_BLOCK FB_TempSimu
VAR_INPUT
	fY: LREAL;
	tCycleTIme: TIME;
	bNoise: BOOL;
END_VAR
VAR_OUTPUT
	fX: LREAL;
END_VAR
VAR
	fbTempSimu: FB_CTRL_PT2;
	SimuPara: ST_CTRL_PT2_PARAMS;
	fbNoiseGen: FB_CTRL_NOISE_GENERATOR;
	tT1: TIME := T#10S;
	tT2: TIME := T#0MS;
	NoisePara: ST_CTRL_NOISE_GENERATOR_PARAMS;
END_VAR

(* 该功能块使用一个二阶系统作为温度模型 *)


SimuPara.fKp := 0.2;
SimuPara.tCtrlCycleTime := tCycleTIme;
SimuPara.tTaskCycleTime := tCycleTIme;
SimuPara.tT1 := tT1;
SimuPara.tT2 := tT2;

NoisePara.fAmplitude := 5;
NoisePara.tCtrlCycleTime := tCycleTIme;
NoisePara.tTaskCycleTime := tCycleTIme;

fbTempSimu(
	fIn:= fY, 
	fManValue:= , 
	eMode:= eCTRL_MODE_ACTIVE, 
	bHold:= , 
	fOut=> , 
	eState=> , 
	eErrorId=> , 
	bError=> , 
	stParams:= SimuPara);
fbNoiseGen(
	fManSyncValue:= 0.0, 
	eMode:= eCTRL_MODE_ACTIVE, 
	fOut=> , 
	eState=> , 
	eErrorId=> , 
	bError=> , 
	stParams:= NoisePara);

IF bNoise THEN
	fX := fbTempSimu.fOut * 10 + 0.005*fbNoiseGen.fOut;
ELSE
	fX := fbTempSimu.fOut * 10;
END_IF;

END_FUNCTION_BLOCK

// ---- TF05Motion/SimpleAxis/FB_SimpleAxis.TcPOU
FUNCTION_BLOCK FB_SimpleAxis
VAR_INPUT
	bPower : BOOL;
	bMovePos : BOOL;
	bMoveVelo : BOOL;
	eMoveMode : E_MoveMode;
	TargetPostion : LREAL;
	TargetVelocity : LREAL;
	bJogFor : BOOL;
	bJogBack : BOOL;
	JogSpeed : LREAL;
	bHome : BOOL;
	bReset : BOOL;
	bStop : BOOL;
	fbAxisSettings : ST_AxisSettings;
END_VAR
VAR_OUTPUT
	(* AxisData *)
	ActPos : LREAL;
	ActVelo : LREAL;
	ModPos : LREAL;
	(* AxisState *)
	NotMoving : BOOL;
	Accelerating : BOOL;
	Moving : BOOL;
	Decelerating : BOOL;
	(* ControlState *)
	PowerOn : BOOL;
	Standstill : BOOL;
	AxisErrID : UDINT;

	(* Fb *)
	bBusy : BOOL;
	bDone : BOOL;
	bAborted : BOOL;
	bError : BOOL;
	nErrID : UDINT;
END_VAR
VAR
	(* Axis *)
	Axis : AXIS_REF;

	
	(* fbCall *)
	mcPower : MC_Power;
	mcMoveAbs : MC_MoveAbsolute;
	mcMoveAbs2 : MC_MoveAbsolute;
	mcMoveMod : MC_MoveModulo;
	mcMoveRel : MC_MoveRelative;
	mcMoveVel : MC_MoveVelocity;
	mcJog : MC_Jog;
	mcReset : MC_Reset;
	mcStop : MC_Stop;

	mcStepAbsSwh : MC_StepAbsoluteSwitch;
	mcFinishHome : MC_FinishHoming;
	
	(* StateMachine *)
	eFbState : E_SimpleAxisState;
	rTrigCommand : R_TRIG;
	(* MoveAbs *)

	ParaPosInPos : LREAL;
	ParaVeloInPos : LREAL;
	(* MoveVelo *)
	ParaVeloInVelo : LREAL;
	(* Jog *)
	ParaJogSpeed : LREAL;
	(* Home *)
	HomingPara : MC_HomingParameter;
	Homed : BOOL;
	HomeRefSignal: MC_Ref_Signal_Ref;
	HomeOptions: ST_Home_Options4;
	HomeDirection: MC_Home_Direction;
	HomeSwhMode: MC_Switch_Mode;
	
	FinishHomeOptions: ST_Home_Options2;
END_VAR

_fbCall();

	(* AxisData *)
ActPos := Axis.NcToPlc.ActPos;
ActVelo := Axis.NcToPlc.ActVelo;
ModPos := Axis.NcToPlc.ModuloActPos;

	(* AxisState *)
NotMoving := Axis.Status.NotMoving;
Accelerating := Axis.Status.Accelerating;
Moving := Axis.Status.HasJob;
Decelerating := Axis.Status.Decelerating;

	(* ControlState *)
Standstill := Axis.Status.StandStill;
AxisErrID := Axis.NcToPlc.ErrorCode;

_CyclicLogic();

METHOD PRIVATE _CyclicLogic : BOOL
VAR_INPUT
END_VAR
rTrigCommand(CLK:= bHome OR bMovePos OR bMoveVelo OR (bJogFor OR bJogBack), Q=> );

CASE eFbState OF
E_SimpleAxisState.Waiting:
	bBusy := FALSE;
	bError := FALSE;
	IF rTrigCommand.Q AND mcPower.Status THEN
		bBusy := TRUE;
		bDone := FALSE;
		bAborted := FALSE;
		bError := FALSE;
		nErrID := 0;
		IF bhome AND NOT Homed THEN
			eFbState := E_SimpleAxisState.BeforeHoming;
		ELSIF bMoveVelo AND Homed THEN
			eFbState := E_SimpleAxisState.BeforeMoveVelo;
		ELSIF bMovePos AND Homed THEN
			eFbState := E_SimpleAxisState.BeforeMovePos;
		ELSIF (bJogFor OR bJogBack) AND Homed THEN
			eFbState := E_SimpleAxisState.BeforeJog;
		END_IF
	END_IF
	
E_SimpleAxisState.BeforeJog:
	ParaJogSpeed := JogSpeed;
	eFbState := E_SimpleAxisState.Joging;
	
E_SimpleAxisState.Joging:
	mcJog.JogForward := bJogFor;
	mcJog.JogBackwards := bJogBack;
	mcJog.Velocity := ParaJogSpeed;
	mcJog(Axis:= Axis);
	IF NOT bJogFor AND NOT bJogBack THEN
		mcJog(Axis:= Axis, JogForward:= FALSE, JogBackwards:= FALSE);
		eFbState := E_SimpleAxisState.JogDone;
	ELSIF mcJog.CommandAborted THEN
		mcJog(Axis:= Axis, JogForward:= FALSE, JogBackwards:= FALSE);
		eFbState := E_SimpleAxisState.Aborted;
	ELSIF mcMoveAbs.Error THEN
		bError := TRUE;
		nErrID := mcMoveAbs.ErrorID;
		mcJog(Axis:= Axis, JogForward:= FALSE, JogBackwards:= FALSE);
		eFbState := E_SimpleAxisState.Error;
	END_IF
	
E_SimpleAxisState.JogDone:
	bDone := TRUE;
	IF Axis.Status.StandStill THEN
		eFbState := E_SimpleAxisState.Waiting;
	END_IF

E_SimpleAxisState.BeforeMovePos:
	ParaPosInPos := TargetPostion;
	ParaVeloInPos := TargetVelocity;
	CASE eMoveMode OF
	E_MoveMode.NotMove:
		eFbState := E_SimpleAxisState.Waiting;
		
	E_MoveMode.MoveAbs:
		eFbState := E_SimpleAxisState.MovingAbs;
		
	E_MoveMode.MoveMod:
		eFbState := E_SimpleAxisState.MovingMod;
		
	E_MoveMode.MoveRel:
		eFbState := E_SimpleAxisState.MovingRel;
	
	END_CASE

E_SimpleAxisState.MovingAbs:
	mcMoveAbs.Position := ParaPosInPos;
	mcMoveAbs.Velocity := ParaVeloInPos;
	mcMoveAbs(Axis := Axis, Execute := TRUE);
	IF mcMoveAbs.Done  THEN
		mcMoveAbs(Axis := Axis, Execute := FALSE);
		eFbState := E_SimpleAxisState.MovePosDone;
	ELSIF mcMoveAbs.CommandAborted THEN
		mcMoveAbs(Axis := Axis, Execute := FALSE);
		eFbState := E_SimpleAxisState.Aborted;
	ELSIF mcMoveAbs.Error THEN
		bError := TRUE;
		nErrID := mcMoveAbs.ErrorID;
		mcMoveAbs(Axis := Axis, Execute := FALSE);
		eFbState := E_SimpleAxisState.Error;
	END_IF
	

E_SimpleAxisState.MovingMod:
	;

E_SimpleAxisState.MovingRel:
	;
E_SimpleAxisState.MovePosDone:
	bDone := TRUE;
	IF Axis.Status.StandStill THEN
		eFbState := E_SimpleAxisState.Waiting;
	END_IF
	
E_SimpleAxisState.BeforeMoveVelo:
	ParaVeloInVelo := TargetVelocity;
	eFbState := E_SimpleAxisState.MovingVelo;

E_SimpleAxisState.MovingVelo:
	mcMoveVel.Velocity := ParaVeloInVelo;
	mcMoveVel(Axis := Axis, Execute := TRUE);
	IF NOT bMoveVelo THEN
		mcMoveVel(Axis := Axis, Execute := FALSE);
		eFbState := E_SimpleAxisState.MoveVeloStop;
	ELSIF mcMoveVel.CommandAborted THEN
		mcMoveVel(Axis := Axis, Execute := FALSE);
		eFbState := E_SimpleAxisState.Aborted;
	ELSIF mcMoveVel.Error THEN
		bError := TRUE;
		nErrID := mcMoveVel.ErrorID;
		mcMoveVel(Axis := Axis, Execute := FALSE);
		eFbState := E_SimpleAxisState.Error;
	END_IF
E_SimpleAxisState.MoveVeloStop:
	mcStop(Axis := Axis, Execute := TRUE);
	IF mcStop.Done AND Axis.Status.HasBeenStopped THEN
		eFbState := E_SimpleAxisState.MoveVeloDone;
	END_IF
	
E_SimpleAxisState.MoveVeloDone:
	bDone := TRUE;
	IF Axis.Status.StandStill THEN
		eFbState := E_SimpleAxisState.Waiting;
	END_IF

	
E_SimpleAxisState.BeforeHoming:
	eFbState := E_SimpleAxisState.Homing;
	
E_SimpleAxisState.Homing:
	mcStepAbsSwh(Axis := Axis, Parameter := HomingPara, Execute := TRUE);
	IF mcStepAbsSwh.Done  THEN
		mcStepAbsSwh(Axis := Axis, Parameter := HomingPara, Execute := FALSE);
		eFbState := E_SimpleAxisState.FinishHoming;
	ELSIF mcStepAbsSwh.CommandAborted THEN
		mcStepAbsSwh(Axis := Axis, Parameter := HomingPara, Execute := FALSE);
		eFbState := E_SimpleAxisState.Aborted;
	ELSIF mcStepAbsSwh.Error THEN
		bError := TRUE;
		nErrID := mcStepAbsSwh.ErrorID;
		mcStepAbsSwh(Axis := Axis, Parameter := HomingPara, Execute := FALSE);
		eFbState := E_SimpleAxisState.Error;
	END_IF

E_SimpleAxisState.FinishHoming:	
	mcFinishHome(Axis := Axis, Parameter := HomingPara, Execute := TRUE);
	IF mcFinishHome.Done  THEN
		mcFinishHome(Axis := Axis, Parameter := HomingPara, Execute := FALSE);
		eFbState := E_SimpleAxisState.HomeToZero;
	ELSIF mcFinishHome.CommandAborted THEN
		mcFinishHome(Axis := Axis, Parameter := HomingPara, Execute := FALSE);
		eFbState := E_SimpleAxisState.Aborted;
	ELSIF mcFinishHome.Error THEN
		bError := TRUE;
		nErrID := mcFinishHome.ErrorID;
		mcFinishHome(Axis := Axis, Parameter := HomingPara, Execute := FALSE);
		eFbState := E_SimpleAxisState.Error;
	END_IF

E_SimpleAxisState.HomeToZero:
	mcMoveAbs.Position := fbAxisSettings.HomeSetpos;
	mcMoveAbs.Velocity := fbAxisSettings.HomeVelo;
	mcMoveAbs(Axis := Axis, Execute := TRUE);
	IF mcMoveAbs.Done  THEN
		mcMoveAbs(Axis := Axis, Execute := FALSE);
		eFbState := E_SimpleAxisState.HomeDone;
	ELSIF mcMoveAbs.CommandAborted THEN
		mcMoveAbs(Axis := Axis, Execute := FALSE);
		eFbState := E_SimpleAxisState.Aborted;
	ELSIF mcMoveAbs.Error THEN
		bError := TRUE;
		nErrID := mcMoveAbs.ErrorID;
		mcMoveAbs(Axis := Axis, Execute := FALSE);
		eFbState := E_SimpleAxisState.Error;
	END_IF
	
E_SimpleAxisState.HomeDone:
	Homed := TRUE;
	bDone := TRUE;
	IF Axis.Status.StandStill THEN
		eFbState := E_SimpleAxisState.Waiting;
	END_IF


E_SimpleAxisState.Aborted:
	bAborted := TRUE;
	IF Axis.Status.StandStill THEN
		eFbState := E_SimpleAxisState.Waiting;
	END_IF


E_SimpleAxisState.Error:
	bError := TRUE;
	IF Axis.Status.StandStill THEN
		eFbState := E_SimpleAxisState.Waiting;
	END_IF
END_CASE
END_METHOD

METHOD PRIVATE _fbCall : BOOL
VAR_INPUT
END_VAR

VAR


END_VAR
Axis.ReadStatus();

mcPower(
	Axis:= Axis, 
	Enable:= bPower, 
	Enable_Positive:= TRUE, 
	Enable_Negative:= TRUE, 
	Override:= 100, 
	BufferMode:= , 
	Options:= , 
	Status=> PowerOn, 
	Busy=> , 
	Active=> , 
	Error=> , 
	ErrorID=> );


mcMoveAbs(
	Axis:= Axis, 
	Execute:= , 
	Position:= , 
	Velocity:= , 
	Acceleration:= fbAxisSettings.MovePosAcc, 
	Deceleration:= fbAxisSettings.MovePosDec, 
	Jerk:= fbAxisSettings.MovePosJerk, 
	BufferMode:= , 
	Options:= , 
	Done=> , 
	Busy=> , 
	Active=> , 
	CommandAborted=> , 
	Error=> , 
	ErrorID=> );





mcMoveMod(
	Axis:= Axis, 
	Execute:= , 
	Position:= , 
	Velocity:= , 
	Acceleration:= fbAxisSettings.MovePosAcc, 
	Deceleration:= fbAxisSettings.MovePosDec, 
	Jerk:= fbAxisSettings.MovePosJerk, 
	Direction:= , 
	BufferMode:= , 
	Options:= , 
	Done=> , 
	Busy=> , 
	Active=> , 
	CommandAborted=> , 
	Error=> , 
	ErrorID=> );
	


mcMoveRel(
	Axis:= Axis, 
	Execute:= , 
	Distance:= , 
	Velocity:= , 
	Acceleration:= fbAxisSettings.MovePosAcc, 
	Deceleration:= fbAxisSettings.MovePosDec, 
	Jerk:= fbAxisSettings.MovePosJerk, 
	BufferMode:= , 
	Options:= , 
	Done=> , 
	Busy=> , 
	Active=> , 
	CommandAborted=> , 
	Error=> , 
	ErrorID=> );
	


mcMoveVel(
	Axis:= Axis, 
	Execute:= , 
	Velocity:= , 
	Acceleration:= fbAxisSettings.MoveVeloAcc, 
	Deceleration:= fbAxisSettings.MoveVeloDec, 
	Jerk:= fbAxisSettings.MoveVeloJerk, 
	Direction:= fbAxisSettings.MoveVeloDirection, 
	BufferMode:= , 
	Options:= , 
	InVelocity=> , 
	Busy=> , 
	Active=> , 
	CommandAborted=> , 
	Error=> , 
	ErrorID=> );
	


mcJog(
	Axis:= Axis, 
	JogForward:= , 
	JogBackwards:= , 
	Mode:= MC_JOGMODE_CONTINOUS, 
	Position:= , 
	Velocity:= , 
	Acceleration:= fbAxisSettings.JogAcc, 
	Deceleration:= fbAxisSettings.JogDec, 
	Jerk:= fbAxisSettings.JogJerk, 
	Done=> , 
	Busy=> , 
	Active=> , 
	CommandAborted=> , 
	Error=> , 
	ErrorID=> );

(*
- (负极限)======>======(原点)=======>=====(正极限) +
回原通过以下两个参数设置, 在当前设置下:
1. 在负极限与原点之间
	向负方向运动直到触发负极限后向正方向运动，经过原点后以原点信号下降沿作为原点
2. 在原点上与1相同
	向负方向运动直到触发负极限后向正方向运动，经过原点后以原点信号下降沿作为原点
3. 在原点与正极限之间
	向负方向运动触发原点后向正方向运动，经过原点后以原点信号下降沿作为原点
*)
HomeDirection := MC_Home_Direction.mcNegativeDirection;
HomeSwhMode := MC_Switch_Mode.mcFallingEdgeInverse;

HomeOptions.DisableDriveAccess := TRUE;
HomeRefSignal.Level := fbAxisSettings.HomeSignal;
mcStepAbsSwh(
	Axis:= Axis, 
	Parameter:= HomingPara, 
	Execute:= , 
	Direction:= HomeDirection, 
	SwitchMode:= HomeSwhMode, 
	ReferenceSignal:= HomeRefSignal, 
	Velocity:= fbAxisSettings.HomeVelo, 
	Acceleration:= fbAxisSettings.HomeAcc, 
	Deceleration:= fbAxisSettings.HomeDec, 
	Jerk:= fbAxisSettings.HomeJerk, 
	SetPosition:= fbAxisSettings.HomeSetpos, 
	TimeLimit:= , 
	DistanceLimit:= , 
	TorqueLimit:= , 
	PositiveLimitSwitch:= fbAxisSettings.HomePosLimit, 
	NegativeLimitSwitch:= fbAxisSettings.HomeNegLimit, 
	BufferMode:= , 
	Options:= HomeOptions, 
	Done=> , 
	Busy=> , 
	Active=> , 
	CommandAborted=> , 
	Error=> , 
	ErrorID=> );	

FinishHomeOptions.DisableDriveAccess := TRUE;
mcFinishHome(
	Axis:= Axis, 
	Parameter:= HomingPara, 
	Execute:= , 
	Distance:= 0, 
	Velocity:= fbAxisSettings.HomeVelo, 
	Acceleration:= fbAxisSettings.HomeAcc, 
	Deceleration:= fbAxisSettings.HomeDec, 
	Jerk:= fbAxisSettings.HomeJerk, 
	BufferMode:= , 
	Options:= FinishHomeOptions, 
	Done=> , 
	Busy=> , 
	CommandAborted=> , 
	Error=> , 
	ErrorID=> );

	
	
mcReset(
	Axis:= Axis, 
	Execute:= bReset, 
	Done=> , 
	Busy=> , 
	Error=> , 
	ErrorID=> );
	


mcStop(
	Axis:= Axis, 
	Execute:= bStop, 
	Deceleration:= , 
	Jerk:= , 
	Options:= , 
	Done=> , 
	Busy=> , 
	Active=> , 
	CommandAborted=> , 
	Error=> , 
	ErrorID=> );
END_METHOD

END_FUNCTION_BLOCK

// ---- TF06Connectivity/TCPIP/FB_TcpSendReceive.TcPOU
FUNCTION_BLOCK FB_TcpSendReceive
VAR_INPUT
	bEnable : BOOL; //启用
	bReset : BOOL;
	sRemoteIp : T_IPv4Addr;
	nRemotePort : UDINT;
	bExecute : BOOL;
	pSendData : POINTER TO BYTE;
	nSendSize : UDINT;
	pRecvData : POINTER TO BYTE;
	nRecvSize : UDINT;
END_VAR
VAR_OUTPUT
	bConnected : BOOL;
	bBusy : BOOL;
	bError : BOOL;
	nRecvByte : UDINT;
END_VAR
VAR
	//功能块调用
	fbConnect : FB_SocketConnect;
	fbClose : FB_SocketClose;
	fbSend : FB_SocketSend;
	fbRecv : FB_SocketReceive;
	
	//状态流转
	stepSendRecv :UDINT;
	
	//连接部分
	tonReconnect : TON;
	hSocket : T_HSOCKET;
	
	//数据收发
	rTrigExecute : R_TRIG;
	tempData : ARRAY[0..255] OF BYTE;
	tonRecvTimeout : TON;
	_AlreadyRecvdData: BOOL;
END_VAR

//主逻辑
_CyclicLogic();

METHOD _CyclicLogic : BOOL
VAR_INPUT
END_VAR

VAR
	
END_VAR
rTrigExecute(CLK:= bExecute, Q=> );
tonReconnect(IN:= , PT:= T#3S, Q=> , ET=> );
tonRecvTimeout(IN:= , PT:= T#3S, Q=> , ET=> );
CASE stepSendRecv OF
	0: //初始状态，等待TCP连接
	fbConnect(bExecute:= FALSE);
	tonReconnect.IN := FALSE;
	IF bEnable AND sRemoteIp <> '' AND nRemotePort <> 0 THEN
		stepSendRecv := 10;
	END_IF

	10: //连接中
	fbConnect(sRemoteHost:= sRemoteIp, nRemotePort:= nRemotePort, bExecute:= TRUE);
	IF fbConnect.bBusy THEN
		;
	ELSE
		IF NOT fbConnect.bError AND (fbConnect.hSocket.handle <> 0) THEN
			hSocket := fbConnect.hSocket;
			stepSendRecv := 20;
		ELSE
			stepSendRecv := 12;
		END_IF
	END_IF

	12: //重连等待
	tonReconnect.IN := TRUE;
	IF tonReconnect.Q THEN
		stepSendRecv := 0;
		tonReconnect.IN := FALSE;
	END_IF

	20: //连接完成
	fbSend(bExecute:= FALSE);
	fbRecv(bExecute:= FALSE);
	tonRecvTimeout.IN := FALSE;
	IF rTrigExecute.Q THEN
		stepSendRecv := 32;
		MEMSET(destAddr:= ADR(pRecvData), fillByte:= 0, n:= nRecvSize);
	END_IF
	
	30://如果触发重收，重收之前的复位
	fbRecv(bExecute:= FALSE);
	stepSendRecv := 32;
	
	32: //先接收，直到收不到为止，防止之前的报文影响
	fbRecv(hSocket:= hSocket, cbLen:= SIZEOF(tempData), pDest:= ADR(tempData), bExecute:= TRUE);
	IF fbRecv.bBusy THEN
		;
	ELSE
		IF fbRecv.bError  THEN
			stepSendRecv := 20; //如果报错，直接取消本次流程，跳到发送前
		ELSE
			IF fbRecv.nRecBytes = 0 THEN
				stepSendRecv := 42; //如果确定之前没有数据接收了，就跳到下一步，开始发送流程
			ELSE
				stepSendRecv := 30; //否则再次尝试接收，直到再也收不到数据
			END_IF
		END_IF
	END_IF
	
	40: //发送，这一步是给重发准备的，目前用不上
	fbSend(bExecute:= FALSE);
	stepSendRecv := 42;
	
	42: //发送
	fbRecv(bExecute:= FALSE);
	fbSend(hSocket:= hSocket, cbLen:= nSendSize, pSrc:= pSendData, bExecute:= TRUE);
	IF fbSend.bBusy THEN
		;
	ELSE
		IF fbSend.bError THEN
			stepSendRecv := 20; //如果报错，直接取消本次流程，跳到发送前
		ELSE
			stepSendRecv := 52;
		END_IF
	END_IF
	
	50://如果触发重收，重收之前的复位
	fbRecv(bExecute:= FALSE);
	stepSendRecv := 52;
	
	52: //接收
	fbSend(bExecute:= FALSE);
	fbRecv(hSocket:= hSocket, cbLen:= nRecvSize, pDest:= pRecvData, bExecute:= TRUE);
	IF fbRecv.bBusy THEN
		;
	ELSE
		IF fbRecv.bError THEN
			stepSendRecv := 20; //如果报错，直接取消本次流程，跳到发送前
		ELSE
			
			IF fbRecv.nRecBytes <>0 THEN
				_AlreadyRecvdData := TRUE;
				stepSendRecv := 50; //收到数据也进入重收
			ELSE
				tonRecvTimeout.IN := TRUE;
				IF _AlreadyRecvdData THEN
					stepSendRecv := 20; //收到数据，就结束流程
					_AlreadyRecvdData := FALSE;
				ELSIF tonRecvTimeout.Q THEN
					stepSendRecv := 20; //如果没收到数据，并且到达了超时时间，就取消流程
				ELSE
					stepSendRecv := 50; //如果没收到数据，且未到超时时间，就进入重收流程
				END_IF
			END_IF
			
		END_IF
	END_IF
	
	
	
END_CASE
END_METHOD

END_FUNCTION_BLOCK

// ---- TF06Connectivity/TCPIP/FB_TcpSendReceiving.TcPOU
(* 2024011902:增加了日志功能 *)
{attribute 'hide_all_locals'}
FUNCTION_BLOCK FB_TcpSendReceiving
VAR_INPUT
	bEnable : BOOL; //启用
	bReset : BOOL; //复位
	sRemoteIp : T_IPv4Addr; //IP地址，如192.168.0.1
	nRemotePort : UDINT; //端口号，如60000
	bExecute : BOOL; //发送触发
	pSendData : POINTER TO BYTE; //发送数据起始地址
	nSendSize : UDINT; //发送数据大小
	pRecvData : POINTER TO BYTE; //接受数据起始地址
	nRecvSize : UDINT; //接受数据大小
END_VAR
VAR_OUTPUT
	bBusyConnect : BOOL;
	bConnected : BOOL;
	bBusySend : BOOL;
	bSendDone : BOOL;
	bBusyRecv : BOOL;
	bRecvDone : BOOL;
	bError : BOOL;
	nRecvBytes : UDINT;
	bDataReceived : BOOL;
END_VAR
VAR
	//功能块调用
	fbConnect : FB_SocketConnect;
	fbClose : FB_SocketClose;
	fbSend : FB_SocketSend;
	fbRecv : FB_SocketReceive;
	
	//状态流转
	stepSendRecv :UDINT;
	stepReceiving : UDINT;
	stepSend : UDINT;
	
	//连接部分
	tonReconnect : TON;
	hSocket : T_HSOCKET;
	
	//数据收发
	rTrigSend : R_TRIG;
	
	tonRecv : TON;
	tempData : ARRAY[0..MAXBUFFERSIZE] OF BYTE;
	hr: BOOL;
	nCountRecvErr : UDINT;

END_VAR

VAR CONSTANT
	MAXBUFFERSIZE: DINT := 1023;
	EmptyhSocket : T_HSOCKET := (handle := 0);
END_VAR

(* 2024011901:TCP收发功能块，单次发，一直收 *)
(* 2024011902:增加了日志功能 *)
IF pSendData = 0 OR pRecvData = 0  THEN
	RETURN;
END_IF
//主逻辑
_CyclicLogic();

METHOD PRIVATE _CyclicLogic : BOOL
VAR_INPUT
END_VAR
VAR

END_VAR

tonReconnect(IN:= , PT:= T#3S, Q=> , ET=> );
bBusyConnect := (stepSendRecv <> 20);
bConnected := (stepSendRecv = 20);
bError := fbConnect.bError OR fbClose.bError OR fbSend.bError OR fbRecv.bError;

CASE stepSendRecv OF
	0: //初始状态，等待TCP连接
	fbConnect(bExecute:= FALSE);
	fbClose(bExecute:= FALSE);
	fbSend(bExecute:= FALSE);
	fbRecv(bExecute := FALSE);
	tonReconnect.IN := FALSE;
	nCountRecvErr := 0;
	IF bEnable AND sRemoteIp <> '' AND nRemotePort <> 0 THEN
		stepSendRecv := 10;
	END_IF

	10: //连接中
	fbConnect(sRemoteHost:= sRemoteIp, nRemotePort:= nRemotePort, bExecute:= TRUE);
	IF fbConnect.bBusy THEN
		;
	ELSE
		IF NOT fbConnect.bError AND (fbConnect.hSocket.handle <> 0) THEN
			hSocket := fbConnect.hSocket;
			stepSendRecv := 20;
			_LogMsg(Level:=0, LogEvent:=FALSE, Msg:= 'Connected', hSocket:= hSocket);
		ELSE
			stepSendRecv := 12;
		END_IF
	END_IF

	12: //重连等待
	tonReconnect.IN := TRUE;
	IF tonReconnect.Q THEN
		_LogMsg(Level:=2, LogEvent:=FALSE, Msg:= 'Connect Failed, Reconnecting', hSocket:= hSocket);
		stepSendRecv := 0;
		tonReconnect.IN := FALSE;
	END_IF

	20: //连接完成
	_Send();
	hr := _Receiving(200,6);
	IF hr = TRUE THEN
		stepSendRecv := 30;
	END_IF
	
	
	30:
	fbClose(hSocket:= hSocket, bExecute:= TRUE );
	IF fbClose.bBusy THEN
		;
	ELSE
		_LogMsg(Level:=2, LogEvent:=FALSE, Msg:= 'Receive Error And Socket Closed', hSocket:= hSocket);
		hSocket := EmptyhSocket;
		stepSendRecv := 0;
	END_IF
END_CASE
END_METHOD

METHOD PRIVATE _LogMsg : BOOL
VAR_INPUT
	Level : INT;
	LogEvent : BOOL;
	Msg : T_MaxString;
	hSocket : T_HSOCKET;
END_VAR
VAR
	TcpInfo : T_MaxString;
	MsgType: DWORD;
	ifLog : DWORD;
	Mask : DWORD;
END_VAR
Msg := CONCAT(STR1:= Msg, STR2:= ', %s');
TcpInfo := 'Handle:';
TcpInfo := CONCAT(STR1:= TcpInfo, STR2:= TO_STRING(hSocket.handle));
TcpInfo := CONCAT(STR1:= TcpInfo, STR2:= ', Ip:');
TcpInfo := CONCAT(STR1:= TcpInfo, STR2:= TO_STRING(hSocket.remoteAddr.sAddr));
TcpInfo := CONCAT(STR1:= TcpInfo, STR2:= ', Port:');
TcpInfo := CONCAT(STR1:= TcpInfo, STR2:= TO_STRING(hSocket.remoteAddr.nPort));
TcpInfo := CONCAT(STR1:= TcpInfo, STR2:= ', AtPort:');
TcpInfo := CONCAT(STR1:= TcpInfo, STR2:= TO_STRING(hSocket.localAddr.nPort));
ifLog := SEL(LogEvent,16#0,ADSLOG_MSGTYPE_LOG);
CASE Level OF
0:
	MsgType := ADSLOG_MSGTYPE_HINT;
1:
	MsgType := ADSLOG_MSGTYPE_WARN;
2:
	MsgType := ADSLOG_MSGTYPE_ERROR;
ELSE
	MsgType := ADSLOG_MSGTYPE_HINT;
END_CASE
Mask := MsgType OR ifLog;
ADSLOGSTR(msgCtrlMask:= Mask, msgFmtStr:= Msg, strArg:= TcpInfo);
END_METHOD

METHOD PRIVATE _Receiving : BOOL
VAR_INPUT
	CycleTime : UDINT;
	ErrorLimit : UDINT;
END_VAR
tonRecv(IN:= , PT:= UDINT_TO_TIME(CycleTime), Q=> , ET=> );
bBusyRecv := (stepReceiving = 10 );
bRecvDone := (stepReceiving <> 10 );
CASE stepReceiving OF
	0:
	bDataReceived := FALSE;
	tonRecv.IN := FALSE;
	fbRecv(bExecute := FALSE);
	stepReceiving := 10;
	
	10:
	
	fbRecv(hSocket:= hSocket, cbLen:= SIZEOF(tempData), pDest:= ADR(tempData), bExecute:= TRUE);
	IF fbRecv.bBusy THEN
		;
	ELSE
		IF fbRecv.bError THEN
			nCountRecvErr := nCountRecvErr + 1;
			_Receiving := (nCountRecvErr > ErrorLimit);
		ELSE
			nCountRecvErr := 0;
			IF fbRecv.nRecBytes <> 0 THEN
				MEMSET(destAddr:= pRecvData, fillByte:= 0, n:= nRecvSize);
				MEMCPY(destAddr:= pRecvData, srcAddr:= ADR(tempData), n:= fbRecv.nRecBytes);
				bDataReceived := TRUE;
			END_IF
			nRecvBytes := fbRecv.nRecBytes;
		END_IF
		stepReceiving := 20;
		tonRecv.IN := TRUE;
	END_IF

	20:
	
	tonRecv.IN := TRUE;
	IF tonRecv.Q THEN
		tonRecv.IN := FALSE;
		stepReceiving := 0;
	END_IF

END_CASE
END_METHOD

METHOD PRIVATE _Reset : BOOL
VAR_INPUT
END_VAR
END_METHOD

METHOD PRIVATE _Send : BOOL
VAR_INPUT
END_VAR
rTrigSend(CLK:= bExecute, Q=> );
bBusySend := (stepSend <> 0);
bSendDone := (stepSend = 0);
CASE stepSend OF
	0:
	fbSend(bExecute:= FALSE);
	IF rTrigSend.Q THEN
		stepSend := 10;

	END_IF
	
	
	10:
	fbSend(hSocket:= hSocket, cbLen:= nSendSize, pSrc:= pSendData, bExecute:= TRUE);
	IF fbSend.bBusy THEN
		;
	ELSE
		IF fbSend.bError THEN
			_Send := TRUE;
		ELSE
			;
		END_IF
		stepSend := 0;
	END_IF
	

END_CASE
END_METHOD

END_FUNCTION_BLOCK

// ---- TF06Connectivity/TCPIP/FB_TcpSendReceivingQueue.TcPOU
//{attribute 'hide_all_locals'}
FUNCTION_BLOCK FB_TcpSendReceivingQueue
VAR_INPUT
	bEnable 			: BOOL; 							//启用
	bReset 				: BOOL; 							//复位,目前设置了自动重连,所以该输入没实现
	sRemoteIp 			: T_IPv4Addr; 						//目标Ip
	nRemotePort 		: UDINT; 							//目标端口
	pRecvData 			: POINTER TO BYTE; 					//接收地址
	nRecvSize 			: UDINT; 							//接收数据区域大小
END_VAR
VAR_OUTPUT
	bBusyConnect 	: BOOL; 								//连接中
	bConnected 		: BOOL; 								//连接完成
	bBusySend 		: BOOL; 								//发送中
	bSendDone 		: BOOL; 								//发送完成
	bBusyRecv 		: BOOL; 								//接受中
	bRecvDone 		: BOOL; 								//接收完成
	bError 			: BOOL; 								//报错
	nRecvBytes 		: UDINT; 								//接收数据长度
	bDataReceived 	: BOOL; 								//接收到数据
END_VAR
VAR
	//功能块调用
	fbConnect : FB_SocketConnect;
	fbClose : FB_SocketClose;
	fbSend : FB_SocketSend;
	fbRecv : FB_SocketReceive;
	fbQueue : FB_SimpleTcpTaskQueue2;
	CurrentTask : ST_TcpTask2;
	//状态流转
	stepSendRecv :UDINT;
	stepReceiving : UDINT;
	stepSend : UDINT;
	//连接部分
	tonReconnect : TON;
	hSocket : T_HSOCKET;
	
	//数据收发
	tonRecv : TON;
	tempData : ARRAY[0..MAXBUFFERSIZE] OF BYTE;
	hr: HRESULT;
	nCountRecvErr : UDINT;

END_VAR

VAR CONSTANT
	MAXBUFFERSIZE: DINT := 1023;
	EmptyhSocket : T_HSOCKET := (handle := 0);
END_VAR

IF pRecvData = 0  THEN
	RETURN;
END_IF
//主逻辑
_CyclicLogic();

METHOD PROTECTED _CyclicLogic : BOOL
VAR_INPUT
END_VAR

VAR
END_VAR
fbQueue();
CurrentTask := fbQueue.CurrentTask;
tonReconnect(IN:= , PT:= T#3S, Q=> , ET=> );
bBusyConnect := (stepSendRecv <> 20);
bConnected := (stepSendRecv = 20);
bError := fbConnect.bError OR fbClose.bError OR fbSend.bError OR fbRecv.bError;

CASE stepSendRecv OF
	0: //初始状态，等待TCP连接
	fbConnect(bExecute:= FALSE);
	fbClose(bExecute:= FALSE);
	fbSend(bExecute:= FALSE);
	fbRecv(bExecute := FALSE);
	tonReconnect.IN := FALSE;
	nCountRecvErr := 0;
	IF bEnable AND sRemoteIp <> '' AND nRemotePort <> 0 THEN
		stepSendRecv := 10;
	END_IF

	10: //连接中
	fbConnect(sRemoteHost:= sRemoteIp, nRemotePort:= nRemotePort, bExecute:= TRUE);
	IF fbConnect.bBusy THEN
		;
	ELSE
		IF NOT fbConnect.bError AND (fbConnect.hSocket.handle <> 0) THEN
			hSocket := fbConnect.hSocket;
			stepSendRecv := 20;
		ELSE
			stepSendRecv := 12;
		END_IF
	END_IF

	12: //重连等待
	tonReconnect.IN := TRUE;
	IF tonReconnect.Q THEN
		stepSendRecv := 0;
		tonReconnect.IN := FALSE;
	END_IF

	20: //连接完成
	_Send();
	hr := _Receiving(200,5); // 接收间隔200ms, 报错限制5次
	IF FAILED(hr) THEN
		stepSendRecv := 30;
	END_IF
	
	
	30:
	fbClose(hSocket:= hSocket, bExecute:= TRUE );
	IF fbClose.bBusy THEN
		;
	ELSE
		hSocket := EmptyhSocket;
		stepSendRecv := 0;
	END_IF
END_CASE
END_METHOD

METHOD PROTECTED _Receiving : HRESULT
VAR_INPUT
	CycleTime : UDINT;
	ErrorLimit : UDINT;
END_VAR
tonRecv(IN:= , PT:= UDINT_TO_TIME(CycleTime), Q=> , ET=> );
bBusyRecv := (stepReceiving = 10 );
bRecvDone := (stepReceiving <> 10 );
CASE stepReceiving OF
	0:
	bDataReceived := FALSE;
	tonRecv.IN := FALSE;
	fbRecv(bExecute := FALSE);
	stepReceiving := 10;
	
	10:
	
	fbRecv(hSocket:= hSocket, cbLen:= SIZEOF(tempData), pDest:= ADR(tempData), bExecute:= TRUE);
	IF fbRecv.bBusy THEN
		;
	ELSE
		IF fbRecv.bError THEN
			nCountRecvErr := nCountRecvErr + 1;
			IF (nCountRecvErr > ErrorLimit) THEN
				_Receiving := -1;
			END_IF
			
		ELSE
			nCountRecvErr := 0;
			IF fbRecv.nRecBytes <> 0 THEN
				MEMSET(destAddr:= pRecvData, fillByte:= 0, n:= nRecvSize);
				MEMCPY(destAddr:= pRecvData, srcAddr:= ADR(tempData), n:= MIN(fbRecv.nRecBytes,nRecvSize) );
				bDataReceived := TRUE;
			END_IF
			nRecvBytes := fbRecv.nRecBytes;
		END_IF
		stepReceiving := 20;
		tonRecv.IN := TRUE;
	END_IF

	20:
	
	tonRecv.IN := TRUE;
	IF tonRecv.Q THEN
		tonRecv.IN := FALSE;
		stepReceiving := 0;
	END_IF

END_CASE
END_METHOD

METHOD PROTECTED _Send : BOOL
VAR_INPUT
END_VAR
bBusySend := (stepSend <> 0);
bSendDone := (stepSend = 0);
CASE stepSend OF
	0:
	fbSend(bExecute:= FALSE);
	IF fbQueue.ActingTaskCount <> 0 THEN
		stepSend := 10;
	END_IF
	
	
	10:
	fbSend(hSocket:= hSocket, cbLen:= CurrentTask.nData, pSrc:= CurrentTask.pData, bExecute:= TRUE);
	IF fbSend.bBusy THEN
		;
	ELSE
		IF fbSend.bError THEN
			_Send := TRUE;
		ELSE
			;
		END_IF
		stepSend := 0;
		fbQueue.FinishTask();
	END_IF
END_CASE
END_METHOD

METHOD AddTask : BOOL
VAR_INPUT
	TaskName : STRING(24);
	TaskType : INT; (* 0:Once, 1:Regular *)
	pData : PVOID;
	nData : UDINT;
END_VAR
fbQueue.AddActingTask(TaskName, TaskType, pData, nData);
END_METHOD

END_FUNCTION_BLOCK

// ---- TF06Connectivity/TCPIP/TcpTaskQueue2/FB_SimpleTcpTaskQueue2.TcPOU
FUNCTION_BLOCK FB_SimpleTcpTaskQueue2
VAR_INPUT
END_VAR
VAR_OUTPUT
END_VAR
VAR
	ActingQueue			: FB_MemRingBufferEx;
	ArrActingQueue		: ARRAY[0..MAXBUFFERSIZE] OF ST_TcpTaskBuffer2;
	
	fbMemMan			: FB_DynMem_Manager2;
	
	PushTask	: ST_TcpTask2;
	PullTask	: ST_TcpTask2;
	EmptyTask	: ST_TcpTask2;
	
	StepTaskConsume : DINT;
	
	_NoTaskToConsume : BOOL;
	_WaitingForTaskDone: BOOL;
	_ActingTaskCount: UDINT;
	_ActingUsedSize: UDINT;
	_ActingFreeSize: UDINT;
END_VAR
VAR CONSTANT
	MAXBUFFERSIZE: UDINT := 128;
END_VAR

_CyclicLogic();

METHOD PROTECTED _CyclicLogic : BOOL
VAR_INPUT
END_VAR
(* 获取队列负载数据 *)
ActingQueue.A_GetFreeSize(pWrite:= , cbWrite:= , pBuffer:= ADR(ArrActingQueue), cbBuffer:= SIZEOF(ArrActingQueue), 
	bOk=> , pRead=> , cbRead=> , nCount=> _ActingTaskCount, cbSize=> _ActingUsedSize, cbFree=> _ActingFreeSize);
(* 状态显示 *)
_NoTaskToConsume := (StepTaskConsume = 0);
_WaitingForTaskDone := (StepTaskConsume <> 0);
(* 如果队列中有事件，取出事件并等待Finish *)
CASE StepTaskConsume OF
	0:
	_NoTaskToConsume := TRUE;
	IF ActingQueue.nCount <> 0 THEN
		StepTaskConsume := 10;
	END_IF
	
	10:
	ActingQueue.A_GetHead(pWrite:= , cbWrite:= , pBuffer:= ADR(ArrActingQueue), cbBuffer:= SIZEOF(ArrActingQueue), 
	bOk=> , pRead=> , cbRead=> , nCount=> _ActingTaskCount, cbSize=> _ActingUsedSize, cbFree=> _ActingFreeSize);
	IF ActingQueue.bOk THEN
		MEMCPY(destAddr:= ADR(PullTask), srcAddr:= ActingQueue.pRead, n:= MIN(SIZEOF(PullTask),ActingQueue.cbRead));
		StepTaskConsume := 20;
	ELSE
		StepTaskConsume := 0;
		ADSLOGSTR(msgCtrlMask:= ADSLOG_MSGTYPE_ERROR OR ADSLOG_MSGTYPE_STRING,
			msgFmtStr:= 'CyclicLogic: FIFO gethead failed', strArg:= '');
	END_IF
	
	20:
	// wait for task done
	
END_CASE
END_METHOD

PROPERTY ActingFreeSize : UDINT
GET
ActingFreeSize := _ActingFreeSize;
END_GET
END_PROPERTY

PROPERTY ActingTaskCount : UDINT
GET
ActingTaskCount := _ActingTaskCount;
END_GET
END_PROPERTY

PROPERTY ActingUsedSize : UDINT
GET
ActingUsedSize := _ActingUsedSize;
END_GET
END_PROPERTY

METHOD AddActingTask : BOOL
VAR_INPUT
	TaskName : STRING(24);
	TaskType : INT; (* 0:Once, 1:Regular *)
	pData : PVOID;
	nData : UDINT;
END_VAR
VAR
	pDynMem : PVOID;
END_VAR
IF nData > ActingQueue.cbFree THEN
	ADSLOGSTR(msgCtrlMask:= ADSLOG_MSGTYPE_ERROR OR ADSLOG_MSGTYPE_STRING,
		msgFmtStr:= 'AddTaskFailed: No free space in FIFO', strArg:= '');
	RETURN;
END_IF
pDynMem := fbMemMan.Alloc(nSize:= nData, bReset:= TRUE);
IF pDynMem = 0 THEN
	ADSLOGSTR(msgCtrlMask:= ADSLOG_MSGTYPE_ERROR OR ADSLOG_MSGTYPE_STRING,
		msgFmtStr:= 'AddTaskFailed: Allocate memory failed', strArg:= '');
	RETURN;
END_IF
MEMCPY(destAddr:= pDynMem, srcAddr:= pData, n:= nData);
PushTask.TaskName := TaskName;
PushTask.TaskType := TaskType;
PushTask.pData := pDynMem;
PushTask.nData := nData;
ActingQueue.A_AddTail(pWrite:= ADR(PushTask), cbWrite:= SIZEOF(PushTask), pBuffer:= ADR(ArrActingQueue), cbBuffer:= SIZEOF(ArrActingQueue), 
	bOk=> AddActingTask, pRead=> , cbRead=> , nCount=> _ActingTaskCount, cbSize=> _ActingUsedSize, cbFree=> _ActingFreeSize);
IF ActingQueue.bOk THEN
	AddActingTask := TRUE;
ELSE
	ADSLOGSTR(msgCtrlMask:= ADSLOG_MSGTYPE_ERROR OR ADSLOG_MSGTYPE_STRING,
		msgFmtStr:= 'AddTaskFailed: FIFO addtail failed ', strArg:= '');
	fbMemMan.Free2(pDynMem);
END_IF
END_METHOD

PROPERTY CurrentTask : ST_TcpTask2
GET
CurrentTask := PullTask;
END_GET
END_PROPERTY

METHOD FinishTask : BOOL
VAR_INPUT
END_VAR
VAR
	pDynMem : PVOID;
END_VAR
(* 调用freehead，释放FIFO头，判断释放是否成功 *)
ActingQueue.A_FreeHead(pWrite:= , cbWrite:= , pBuffer:= ADR(ArrActingQueue), cbBuffer:= SIZEOF(ArrActingQueue), 
	bOk=> , pRead=> , cbRead=> , nCount=> _ActingTaskCount, cbSize=> _ActingUsedSize, cbFree=> _ActingFreeSize);
IF ActingQueue.bOk THEN
	IF ActingQueue.nCount <> 0 THEN
		StepTaskConsume := 10;
	ELSE
		StepTaskConsume := 0;
	END_IF
ELSE
	ADSLOGSTR(msgCtrlMask:= ADSLOG_MSGTYPE_ERROR OR ADSLOG_MSGTYPE_STRING,
		msgFmtStr:= 'FinishTaskFailed: FIFO freehead failed', strArg:= '');
	RETURN;
END_IF

FinishTask := TRUE;
pDynMem := PullTask.pData;
PullTask := EmptyTask;
//MEMCPY(destAddr:= ADR(PullTask), srcAddr:= ADR(EmptyTask), n:= SIZEOF(PullTask));
fbMemMan.Free2(pDynMem);
END_METHOD

PROPERTY NoTaskToConsume : BOOL
GET
NoTaskToConsume := _NoTaskToConsume;
END_GET
END_PROPERTY

PROPERTY WaitingForTaskDone : BOOL
GET
WaitingForTaskDone := _WaitingForTaskDone;
END_GET
END_PROPERTY

END_FUNCTION_BLOCK

// ---- TF06Connectivity/TCPIP/SimpleClient/SimpleTcpClient.TcPOU
FUNCTION_BLOCK SimpleTcpClient
VAR_INPUT
END_VAR
VAR_OUTPUT
END_VAR
VAR
	fbSocketConnect : FB_ClientServerConnection;
	fbSocketSend : FB_SocketSend;
	fbSocketReceive : FB_SocketReceive;
	fbGetLinkStatus: FB_SocketGetLinkStatus;
	tonLinkStatus : TON;
	(* Properties *)
	_SktPara : stSktPara;
	_Connected : BOOL;
	_hSocket : T_HSOCKET;
	_LastRecvBytes : UDINT;
	_Error : BOOL;
	_ErrorID : UDINT;
	_SentCounter : UDINT;
	_SentBytes : UDINT;
	_RecvdCounter : UDINT;
	_RecvdBytes : UDINT;
	(* Connect *)

	StepReconnect : UDINT;
	(* GetLinkStatus *)
	LastStatus : BOOL;
	(* SendReceive *)
	StepSendReceive : UDINT;
	RecvTimes : UDINT;
	(* SendRecv *)
	StepSendRecv : UDINT;
	TryRecvTimes : UDINT;
	TonTryRecvTimeout : TON;
END_VAR

METHOD ClearDiagData : BOOL
VAR_INPUT
END_VAR
_SentCounter :=0 ;
_SentBytes :=0  ;
_RecvdCounter :=0 ;
_RecvdBytes :=0 ;
ClearDiagData := TRUE;
END_METHOD

METHOD Connect : stConnState
VAR_INPUT
	sRemoteHost : T_IPv4Addr;
	nRemotePort : UDINT;
END_VAR

fbSocketConnect.sRemoteHost := sRemoteHost;
fbSocketConnect.nRemotePort := nRemotePort;
fbSocketConnect.bEnable := TRUE;
fbSocketConnect(sSrvNetID:= '', nMode:= 16#8000_0000, sRemoteHost:= , nRemotePort:= , bEnable:= , tReconnect:= T#45S, 
	bBusy=> , bError=> , nErrId=> , hSocket=> , eState=> );

CASE StepReconnect OF
	0:
		IF _SktPara.AutoReconnect = TRUE AND _Connected = TRUE AND  GetLinkStatus() = FALSE THEN
			Reconnect();
			StepReconnect := 10 ;
		END_IF
	10:
		IF  GetLinkStatus() = TRUE THEN
			StepReconnect := 0 ;
		END_IF
END_CASE

(* 返回值 *)
Connect.eState := fbSocketConnect.eState;
Connect.bConnected := (fbSocketConnect.eState = eSOCKET_CONNECTED);
Connect.bError := fbSocketConnect.bError;
Connect.nErrId := fbSocketConnect.nErrId;
Connect.hSocket := fbSocketConnect.hSocket;
(* 内部变量 *)
_Connected := (fbSocketConnect.eState = eSOCKET_CONNECTED);
_hSocket := fbSocketConnect.hSocket;
_Error := fbSocketConnect.bError;
_ErrorID := fbSocketConnect.nErrId;
END_METHOD

PROPERTY PUBLIC Connected : bool
GET
Connected := _Connected;
END_GET
END_PROPERTY

METHOD Disconnect : stConnState
VAR_INPUT
END_VAR
fbSocketConnect.bEnable := FALSE;
fbSocketConnect(sSrvNetID:= '', nMode:= 16#8000_0000, sRemoteHost:= , nRemotePort:= , bEnable:= , tReconnect:= T#45S, 
	bBusy=> , bError=> , nErrId=> , hSocket=> , eState=> );


(* 返回值 *)
Disconnect.eState := fbSocketConnect.eState;
Disconnect.bConnected := (fbSocketConnect.eState <> eSOCKET_DISCONNECTED);
Disconnect.bError := fbSocketConnect.bError;
Disconnect.nErrId := fbSocketConnect.nErrId;
Disconnect.hSocket := fbSocketConnect.hSocket;

(* 内部变量 *)
_Connected := (fbSocketConnect.eState <> eSOCKET_DISCONNECTED);
END_METHOD

PROPERTY Error : bool
GET
Error := _Error;
END_GET
END_PROPERTY

PROPERTY ErrorID : UDINT
GET
ErrorID := _ErrorID;
END_GET
END_PROPERTY

METHOD GetLinkStatus : BOOL
VAR_INPUT
END_VAR
tonLinkStatus(IN:= NOT tonLinkStatus.Q, PT:= T#500MS, Q=> , ET=> );
fbGetLinkStatus.hSocket := _hSocket;
fbGetLinkStatus.bExecute := tonLinkStatus.Q;
fbGetLinkStatus(sSrvNetId:= , hSocket:= , bExecute:= , tTimeout:= , 
	bBusy=> , bError=> , nErrId=> , bLinkError=> );
//GetLinkStatus := NOT fbGetLinkStatus.bBusy AND NOT fbGetLinkStatus.bError AND NOT fbGetLinkStatus.bLinkError;
IF fbGetLinkStatus.bBusy THEN
	GetLinkStatus := LastStatus;
ELSE
	LastStatus := GetLinkStatus := NOT fbGetLinkStatus.bError AND NOT fbGetLinkStatus.bLinkError;
END_IF
END_METHOD

PROPERTY hSocket : T_HSOCKET
GET
hSocket := _hSocket;
END_GET
END_PROPERTY

PROPERTY LastRecvBytes : udint
GET
LastRecvBytes := _LastRecvBytes;
END_GET
END_PROPERTY

METHOD Receive : DINT
VAR_INPUT
	pRecvAdr : POINTER TO BYTE;
	nRecvSize : UDINT;
END_VAR
VAR
	
END_VAR
Receive := 0;
IF pRecvAdr = 0 OR nRecvSize = 0 OR _Connected = FALSE THEN
	RETURN;
ELSE
	fbSocketReceive.hSocket := _hSocket;
	fbSocketReceive.pDest := pRecvAdr;
	fbSocketReceive.cbLen := nRecvSize;
	fbSocketReceive.bExecute := TRUE;
	fbSocketReceive(
		sSrvNetId:= '', 
		hSocket:= , 
		cbLen:= , 
		pDest:= , 
		bExecute:= , 
		tTimeout:= , 
		bBusy=> , 
		bError=> , 
		nErrId=> , 
		nRecBytes=> );
	IF NOT fbSocketReceive.bBusy THEN
		fbSocketReceive(bExecute := FALSE);
		IF NOT fbSocketReceive.bError THEN
			_LastRecvBytes := fbSocketReceive.nRecBytes;
			_RecvdCounter := _RecvdCounter + 1;
			_RecvdBytes := _RecvdBytes + fbSocketReceive.nRecBytes;
			Receive := 1; 
			IF _SktPara.EnableRecvLog = TRUE AND fbSocketReceive.nRecBytes > 0 THEN
				ADSLOGSTR(msgCtrlMask:= ADSLOG_MSGTYPE_LOG, msgFmtStr:= 'RecvMsg : %s', strArg:= UDINT_TO_STRING(fbSocketReceive.nRecBytes));
			END_IF
			
		ELSE
			_Error := fbSocketReceive.bError;
			_ErrorID := fbSocketReceive.nErrId;
			Receive := -2;
		END_IF
			
	END_IF
END_IF
END_METHOD

METHOD Reconnect : BOOL
VAR_INPUT
END_VAR
fbSocketConnect.bEnable := FALSE;
fbSocketConnect();
fbSocketConnect.bEnable := TRUE;
fbSocketConnect();
Reconnect := TRUE;
END_METHOD

PROPERTY RecvdBytes : UDINT
GET
RecvdBytes := _RecvdBytes;
END_GET
SET
_RecvdBytes := RecvdBytes;
END_SET
END_PROPERTY

PROPERTY RecvdCounter : UDINT
GET
RecvdCounter := _RecvdCounter;
END_GET
SET
_RecvdCounter := RecvdCounter;
END_SET
END_PROPERTY

METHOD Send : DINT
VAR_INPUT
	pSendAdr : POINTER TO BYTE;
	nSendSize : UDINT;
END_VAR
Send := 0;
IF pSendAdr = 0 OR nSendSize = 0 OR _Connected = FALSE THEN
	RETURN;
ELSE
	fbSocketSend.hSocket := _hSocket;
	fbSocketSend.pSrc := pSendAdr;
	fbSocketSend.cbLen := nSendSize;
	fbSocketSend.bExecute := TRUE;
	fbSocketSend(
		sSrvNetId:= '', 
		hSocket:= , 
		cbLen:= , 
		pSrc:= , 
		bExecute:= , 
		tTimeout:= , 
		bBusy=> , 
		bError=> , 
		nErrId=> );
	
	IF NOT fbSocketSend.bBusy THEN
		fbSocketSend(bExecute:= FALSE);
		IF NOT fbSocketSend.bError THEN
			Send := 1;
			_SentCounter := _SentCounter + 1;
			_SentBytes := _SentBytes + nSendSize;
			IF _SktPara.EnableSendLog = TRUE THEN
				ADSLOGSTR(msgCtrlMask:= ADSLOG_MSGTYPE_LOG, msgFmtStr:= 'SendBytes : %s', strArg:= UDINT_TO_STRING(nSendSize));
			END_IF
			
		ELSE
			_Error := fbSocketSend.bError;
			_ErrorID := fbSocketSend.nErrId;
			Send := -1;
		END_IF
	END_IF
END_IF
END_METHOD

PROPERTY SendBytes : UDINT
GET
SendBytes := _SentBytes;
END_GET
SET
_SentBytes := SendBytes;
END_SET
END_PROPERTY

PROPERTY SendCounter : UDINT
GET
SendCounter := _SentCounter;
END_GET
SET
_SentCounter := SendCounter;
END_SET
END_PROPERTY

METHOD INTERNAL SendRecive : DINT
VAR_INPUT
	pSendAdr : POINTER TO BYTE;
	nSendSize : UDINT;
	pRecvAdr : POINTER TO BYTE;
	nRecvSize : UDINT;
END_VAR
SendRecive := 0;
IF pSendAdr = 0 OR nSendSize = 0 OR pRecvAdr = 0 OR nRecvSize = 0 OR _Connected = FALSE THEN
	RETURN;
ELSE
	CASE StepSendReceive OF	
	0:
		fbSocketSend.hSocket := _hSocket;
		fbSocketSend.pSrc := pSendAdr;
		fbSocketSend.cbLen := nSendSize;
		fbSocketSend.bExecute := TRUE;
		fbSocketSend();
	
		IF NOT fbSocketSend.bBusy THEN
			fbSocketSend(bExecute:= FALSE);
			IF NOT fbSocketSend.bError THEN
				StepSendReceive := 10;
				_SentCounter := _SentCounter + 1;
				_SentBytes := _SentBytes + nSendSize;
			ELSE
				_Error := fbSocketSend.bError;
				_ErrorID := fbSocketSend.nErrId;
				SendRecive := -1;
				StepSendReceive := 0;
			END_IF
		END_IF

	
	10:
		fbSocketReceive.hSocket := _hSocket;
		fbSocketReceive.pDest := pRecvAdr;
		fbSocketReceive.cbLen := nRecvSize;
		fbSocketReceive.bExecute := TRUE;
		fbSocketReceive();
		IF NOT fbSocketReceive.bBusy THEN
			fbSocketReceive(bExecute := FALSE);
			IF NOT fbSocketReceive.bError THEN
				IF fbSocketReceive.nRecBytes > 0 THEN
					_LastRecvBytes := fbSocketReceive.nRecBytes;
					_RecvdCounter := _RecvdCounter + 1;
					_RecvdBytes := _RecvdBytes + fbSocketReceive.nRecBytes;
					RecvTimes := 0;
					SendRecive := 1;
					StepSendReceive := 0;
				ELSE
					IF RecvTimes > 10 THEN
						SendRecive := -3;
						StepSendReceive := 0;
					ELSE
						RecvTimes := RecvTimes + 1;
					END_IF
				END_IF
			ELSE
				_Error := fbSocketReceive.bError;
				_ErrorID := fbSocketReceive.nErrId;
				SendRecive := -2;
				StepSendReceive := 0;
			END_IF
		END_IF

	//12:
		
		
	END_CASE
END_IF
END_METHOD

METHOD SendRecv : DINT
VAR_INPUT
	pSendAdr : POINTER TO BYTE;
	nSendSize : UDINT;
	pRecvAdr : POINTER TO BYTE;
	nRecvSize : UDINT;
END_VAR
VAR
	hrSend : DINT;
	hrRecv : DINT;
END_VAR
SendRecv := 0;
TonTryRecvTimeout(IN:= , PT:= _SktPara.SendRecvTimeOut, Q=> , ET=> );
IF pSendAdr = 0 OR nSendSize = 0 OR pRecvAdr = 0 OR nRecvSize = 0 OR _Connected = FALSE THEN
	RETURN;
ELSE
	CASE StepSendRecv OF	
	0:
		hrSend := Send(pSendAdr, nSendSize);
		CASE hrSend OF
		1:
			StepSendRecv := 10;
			
		ELSE
			SendRecv := hrSend;
		END_CASE
	10:
		hrRecv := Receive(pRecvAdr, nRecvSize);
		CASE hrRecv OF
		0:
			;
		1:
			IF _LastRecvBytes > 0 THEN
				TryRecvTimes := 0;
				SendRecv := 1;
				TonTryRecvTimeout.IN := FALSE;
				StepSendRecv := 0;
			ELSE
				TonTryRecvTimeout.IN := TRUE;
				IF TonTryRecvTimeout.Q THEN
					SendRecv := -4;
					StepSendRecv := 0;
					TonTryRecvTimeout.IN := FALSE;
				END_IF
			END_IF
			
		ELSE
			SendRecv := hrRecv;
		END_CASE
	//12:
		
		
	END_CASE
END_IF
END_METHOD

PROPERTY SktPara : stSktPara
GET
SktPara := _SktPara;
END_GET
SET
_SktPara := SktPara;
END_SET
END_PROPERTY

END_FUNCTION_BLOCK

// ---- TF06Connectivity/TCPIP/TcpTaskQueue/FB_SimpleTcpTaskQueue.TcPOU
FUNCTION_BLOCK FB_SimpleTcpTaskQueue
VAR_INPUT
END_VAR
VAR_OUTPUT
END_VAR
VAR
	WaitingQueue		: FB_MemRingBufferEx;
	ArrWaitingQueue		: ARRAY[0..MAXBUFFERSIZE] OF ST_TcpTaskBuffer;
	ActingQueue			: FB_MemRingBufferEx;
	ArrActingQueue		: ARRAY[0..MAXBUFFERSIZE] OF ST_TcpTaskBuffer;
	
	PushTask	: ST_TcpTask;
	PopTask		: ST_TcpTask;
	EmptyTask	: ST_TcpTask;
	
	StepTaskConsume : DINT;
	
	_NoTaskToConsume : BOOL;
	_WaitingForTaskDone: BOOL;
	
	_TaskComplete : BOOL;
	
	_WaitingTaskCount: UDINT;
	_WaitingUsedSize: UDINT;
	_WaitingFreeSize: UDINT;
	
	_ActingTaskCount: UDINT;
	_ActingTotalSize: UDINT;
	_ActingFreeSize: UDINT;

END_VAR

VAR CONSTANT
	MAXBUFFERSIZE: UDINT := 128;
END_VAR

WaitingQueue(pWrite:= , cbWrite:= , pBuffer:= ADR(ArrWaitingQueue), cbBuffer:= SIZEOF(ArrWaitingQueue), 
	bOk=> , pRead=> , cbRead=> , nCount=> _WaitingTaskCount, cbSize=> _WaitingUsedSize, cbFree=> _WaitingFreeSize);
ActingQueue(pWrite:= , cbWrite:= , pBuffer:= ADR(ArrActingQueue), cbBuffer:= SIZEOF(ArrActingQueue), 
	bOk=> , pRead=> , cbRead=> , nCount=> _ActingTaskCount, cbSize=> _ActingTotalSize, cbFree=> _ActingFreeSize);

_NoTaskToConsume := (StepTaskConsume = 0);
_WaitingForTaskDone := (StepTaskConsume <> 0);
CASE StepTaskConsume OF
	0:
	_NoTaskToConsume := TRUE;
	IF ActingQueue.nCount <> 0 THEN
		StepTaskConsume := 10;
	END_IF
	
	10:
	ActingQueue.A_GetHead(pWrite:= , cbWrite:= , pBuffer:= ADR(ArrActingQueue), cbBuffer:= SIZEOF(ArrActingQueue), 
	bOk=> , pRead=> , cbRead=> , nCount=> _ActingTaskCount, cbSize=> _ActingTotalSize, cbFree=> _ActingFreeSize);
	IF ActingQueue.bOk THEN
		MEMCPY(destAddr:= ADR(PopTask), srcAddr:= ActingQueue.pRead, n:= MIN(SIZEOF(PopTask),ActingQueue.cbRead));
		_TaskComplete := FALSE;
		StepTaskConsume := 20;
	ELSE
		StepTaskConsume := 0;
	END_IF
	
	20:
	// wait for task done
	
END_CASE

PROPERTY ActingTaskCount : UDINT
GET
ActingTaskCount := _ActingTaskCount;
END_GET
END_PROPERTY

METHOD AddActingTask : BOOL
VAR_INPUT
	TaskName : STRING(24);
	TaskType : INT; (* 0:Once, 1:Regular *)
	TaskData : ARRAY[0..255] OF BYTE;
END_VAR
PushTask.TaskName := TaskName;
PushTask.TaskType := TaskType;
PushTask.TaskData := TaskData;
ActingQueue.A_AddTail(pWrite:= ADR(PushTask), cbWrite:= SIZEOF(PushTask), pBuffer:= ADR(ArrActingQueue), cbBuffer:= SIZEOF(ArrActingQueue), 
	bOk=> AddActingTask, pRead=> , cbRead=> , nCount=> _ActingTaskCount, cbSize=> _ActingTotalSize, cbFree=> _ActingFreeSize);
END_METHOD

PROPERTY CurrentTask : ST_TcpTask
GET
CurrentTask := PopTask;
END_GET
END_PROPERTY

METHOD FinishTask : BOOL
VAR_INPUT
END_VAR
ActingQueue.A_FreeHead(pWrite:= , cbWrite:= , pBuffer:= ADR(ArrActingQueue), cbBuffer:= SIZEOF(ArrActingQueue), 
bOk=> , pRead=> , cbRead=> , nCount=> _ActingTaskCount, cbSize=> _ActingTotalSize, cbFree=> _ActingFreeSize);
IF ActingQueue.bOk THEN
	MEMCPY(destAddr:= ADR(PopTask), srcAddr:= ADR(EmptyTask), n:= SIZEOF(ST_TcpTask));
	IF ActingQueue.nCount <> 0 THEN
		StepTaskConsume := 10;
	ELSE
		StepTaskConsume := 0;
	END_IF
END_IF
END_METHOD

END_FUNCTION_BLOCK

// ---- TF06Connectivity/TCPIP/[obsolete]/FB_TcpSendReceivingHistroy.TcPOU
{attribute 'hide_all_locals'}
FUNCTION_BLOCK FB_TcpSendReceivingHistroy
VAR_INPUT
	bEnable 			: BOOL; 								//启用
	bReset 				: BOOL; 								//复位,目前设置了自动重连,所以该输入没实现
	sRemoteIp 		: T_IPv4Addr; 						//目标Ip
	nRemotePort 		: UDINT; 								//目标端口
	bExecute 			: BOOL; 								//发送
	pSendData 		: POINTER TO BYTE; 			//发送地址
	nSendSize 		: UDINT; 								//发送数据区域大小
	pRecvData 		: POINTER TO BYTE; 			//接收地址
	nRecvSize 			: UDINT; 								//接收数据区域大小
END_VAR
VAR_OUTPUT
	bBusyConnect 	: BOOL; 								//连接中
	bConnected 		: BOOL; 								//连接完成
	bBusySend 		: BOOL; 								//发送中
	bSendDone 		: BOOL; 								//发送完成
	bBusyRecv 		: BOOL; 								//接受中
	bRecvDone 		: BOOL; 								//接收完成
	bError 				: BOOL; 								//报错
	nRecvBytes 		: UDINT; 								//接收数据长度
	bDataReceived 	: BOOL; 								//接收到数据
END_VAR
VAR
	//功能块调用
	fbConnect : FB_SocketConnect;
	fbClose : FB_SocketClose;
	fbSend : FB_SocketSend;
	fbRecv : FB_SocketReceive;
	
	//状态流转
	stepSendRecv :UDINT;
	stepReceiving : UDINT;
	stepSend : UDINT;
	//连接部分
	tonReconnect : TON;
	hSocket : T_HSOCKET;
	
	//数据收发
	rTrigSend : R_TRIG;
	
	tonRecv : TON;
	tempData : ARRAY[0..MAXBUFFERSIZE] OF BYTE;
	hr: BOOL;
	nCountRecvErr : UDINT;

END_VAR

VAR CONSTANT
	MAXBUFFERSIZE: DINT := 1023;
	EmptyhSocket : T_HSOCKET := (handle := 0);
END_VAR


IF pSendData = 0 OR pRecvData = 0  THEN
	RETURN;
END_IF
//主逻辑
_CyclicLogic();

METHOD PRIVATE _CyclicLogic : BOOL
VAR_INPUT
END_VAR

VAR
END_VAR



tonReconnect(IN:= , PT:= T#3S, Q=> , ET=> );
bBusyConnect := (stepSendRecv <> 20);
bConnected := (stepSendRecv = 20);
bError := fbConnect.bError OR fbClose.bError OR fbSend.bError OR fbRecv.bError;

CASE stepSendRecv OF
	0: //初始状态，等待TCP连接
	fbConnect(bExecute:= FALSE);
	fbClose(bExecute:= FALSE);
	fbSend(bExecute:= FALSE);
	fbRecv(bExecute := FALSE);
	tonReconnect.IN := FALSE;
	nCountRecvErr := 0;
	IF bEnable AND sRemoteIp <> '' AND nRemotePort <> 0 THEN
		stepSendRecv := 10;
	END_IF

	10: //连接中
	fbConnect(sRemoteHost:= sRemoteIp, nRemotePort:= nRemotePort, bExecute:= TRUE);
	IF fbConnect.bBusy THEN
		;
	ELSE
		IF NOT fbConnect.bError AND (fbConnect.hSocket.handle <> 0) THEN
			hSocket := fbConnect.hSocket;
			stepSendRecv := 20;
		ELSE
			stepSendRecv := 12;
		END_IF
	END_IF

	12: //重连等待
	tonReconnect.IN := TRUE;
	IF tonReconnect.Q THEN
		stepSendRecv := 0;
		tonReconnect.IN := FALSE;
	END_IF

	20: //连接完成
	_Send();
	hr := _Receiving(200,6);
	IF hr = TRUE THEN
		stepSendRecv := 30;
	END_IF
	
	
	30:
	fbClose(hSocket:= hSocket, bExecute:= TRUE );
	IF fbClose.bBusy THEN
		;
	ELSE
		hSocket := EmptyhSocket;
		stepSendRecv := 0;
	END_IF
END_CASE
END_METHOD

METHOD PRIVATE _Receiving : BOOL
VAR_INPUT
	CycleTime : UDINT;
	ErrorLimit : UDINT;
END_VAR
tonRecv(IN:= , PT:= UDINT_TO_TIME(CycleTime), Q=> , ET=> );
bBusyRecv := (stepReceiving = 10 );
bRecvDone := (stepReceiving <> 10 );
CASE stepReceiving OF
	0:
	bDataReceived := FALSE;
	tonRecv.IN := FALSE;
	fbRecv(bExecute := FALSE);
	stepReceiving := 10;
	
	10:
	
	fbRecv(hSocket:= hSocket, cbLen:= SIZEOF(tempData), pDest:= ADR(tempData), bExecute:= TRUE);
	IF fbRecv.bBusy THEN
		;
	ELSE
		IF fbRecv.bError THEN
			nCountRecvErr := nCountRecvErr + 1;
			_Receiving := (nCountRecvErr > ErrorLimit);
		ELSE
			nCountRecvErr := 0;
			IF fbRecv.nRecBytes <> 0 THEN
				MEMSET(destAddr:= pRecvData, fillByte:= 0, n:= nRecvSize);
				MEMCPY(destAddr:= pRecvData, srcAddr:= ADR(tempData), n:= MIN(fbRecv.nRecBytes,nRecvSize) );
				bDataReceived := TRUE;
			END_IF
			nRecvBytes := fbRecv.nRecBytes;
		END_IF
		stepReceiving := 20;
		tonRecv.IN := TRUE;
	END_IF

	20:
	
	tonRecv.IN := TRUE;
	IF tonRecv.Q THEN
		tonRecv.IN := FALSE;
		stepReceiving := 0;
	END_IF

END_CASE
END_METHOD

METHOD PRIVATE _Send : BOOL
VAR_INPUT
END_VAR
rTrigSend(CLK:= bExecute, Q=> );
bBusySend := (stepSend <> 0);
bSendDone := (stepSend = 0);
CASE stepSend OF
	0:
	fbSend(bExecute:= FALSE);
	IF rTrigSend.Q THEN
		stepSend := 10;

	END_IF
	
	
	10:
	fbSend(hSocket:= hSocket, cbLen:= nSendSize, pSrc:= pSendData, bExecute:= TRUE);
	IF fbSend.bBusy THEN
		;
	ELSE
		IF fbSend.bError THEN
			_Send := TRUE;
		ELSE
			;
		END_IF
		stepSend := 0;
	END_IF
	

END_CASE
END_METHOD

END_FUNCTION_BLOCK

// ---- TF11PlcSystem/AnalogScale/AnalogScale.TcPOU
(* OutputValue := InputValue * (OutputMax - OutputMin)/(InputMax - InputMin) + OutputMin *)
FUNCTION_BLOCK AnalogScale
VAR_INPUT
	InputValue	: LREAL;
	InputMin	: LREAL:=0;
	InputMax	: LREAL:=100;
	OutputMin	: LREAL:=0;
	OutputMax	: LREAL:=100;
END_VAR
VAR_OUTPUT
	OutputValue	: LREAL;
	Percentage : LREAL;
	DataInvalid : BOOL;
END_VAR
VAR
END_VAR

IF InputMax - InputMin = 0 THEN
	DataInvalid := TRUE;
ELSE
	OutputValue := InputValue * (OutputMax - OutputMin)/(InputMax - InputMin) + OutputMin;
	Percentage := (InputValue - InputMin)/(InputMax - InputMin);
	DataInvalid := FALSE;
END_IF

END_FUNCTION_BLOCK

// ---- TF11PlcSystem/AnalogScale/AnalogScaleWithAlarm.TcPOU
(* OutputValue := InputValue * (OutputMax - OutputMin)/(InputMax - InputMin) + OutputMin *)
FUNCTION_BLOCK AnalogScaleWithAlarm
VAR_INPUT
	InputValue	: LREAL;
	InputMin	: LREAL:=0;
	InputMax	: LREAL:=100;
	OutputMin	: LREAL:=0;
	OutputMax	: LREAL:=100;
	LL_Set	: LREAL;
	L_Set	: LREAL;
	H_Set	: LREAL;
	HH_Set	: LREAL;
END_VAR
VAR_OUTPUT
	OutputValue	: LREAL;
	Percentage : LREAL;
	DataInvalid : BOOL;
	LL : BOOL;
	L : BOOL;
	H : BOOL;
	HH : BOOL;
END_VAR
VAR
END_VAR

IF InputMax - InputMin = 0 THEN
	DataInvalid := TRUE;
ELSE
	OutputValue := InputValue * (OutputMax - OutputMin)/(InputMax - InputMin) + OutputMin;
	Percentage := (InputValue - InputMin)/(InputMax - InputMin);
	DataInvalid := FALSE;
END_IF

LL := OutputValue < LL_Set;
L := OutputValue < L_Set;
H := OutputValue > H_Set;
HH := OutputValue > HH_Set;

END_FUNCTION_BLOCK

// ---- TF11PlcSystem/ET_DoubleBuffer/DataFileLogger.TcPOU
{attribute 'no_check' := ''}
//Extension to FB "DoubleBuffer" to write the recorded data cyclic into a file 
{attribute 'enable_dynamic_creation'}
FUNCTION_BLOCK DataFileLogger EXTENDS DoubleBuffer
VAR_OUTPUT CONSTANT 
	{attribute 'displaymode':='binary'}
	OPTION_KEEP_FILE_ON_ERROR								: 	BYTE := 2#0000_0001; //Keep file open in error case to be able to contine after reset
	{attribute 'displaymode':='binary'}
	OPTION_START_WITH_NEW_FILE								: 	BYTE := 2#1000_0000; //Create empty file with enable flag instead open and continue existing file
END_VAR                     								
VAR_INPUT                   								
	Enable													: 	BOOL; //Enable to write looked data cyclic into file  
	ResetTrig												: 	BOOL; //Reset internal error 

{attribute 'displaymode':='binary'}
	Options													: 	BYTE := 2#00000000; // See outputs constant OPTION_xxx
	Path													: 	STRING := 'C:\temp'; //Path and filename
	Filetype												: 	STRING(6) := '.log'; //file tpye
END_VAR                     								
VAR_IN_OUT                  								
END_VAR                     								
VAR_OUTPUT       
	TimeWriteFile											:	TIME; //Elapsed time to write data to file 
	hFile													: 	UINT; //Current file handle
	Busy													: 	BOOL; //Write msg to file active   
	Error													: 	BOOL;     
	{attribute 'displaymode':='hex'}   								
	ErrorId													: 	UDINT; //Ads error Id of file handling function blocks or HRESULT (hr) ADS error code 
END_VAR                     								
VAR            
//local ************************************************************************************
	WriteCounter											:	UDINT; //Endless write counter fyi
	State													: 	INT;
	StartTimeWriteData										:	TIME;			

//trigger *********************************************************************************

//timer ***********************************************************************************

//instances ***********************************************************************************             								
	FILEOPEN												: 	FB_FileOpen := (sNetId:='',tTimeout:=DEFAULT_ADS_TIMEOUT, ePath:=PATH_GENERIC);
	FILECLOSE												: 	FB_FileClose := (sNetId:='',tTimeout:=DEFAULT_ADS_TIMEOUT);
	FILEWRITE												: 	FB_FileWrite := (sNetId:='',tTimeout:=DEFAULT_ADS_TIMEOUT);

//Dummys ****************************************************************************************

END_VAR

	(* Data file logger based on two buffer concept 		*)
	(********************************************************)

(* Sequence started by method addData if buffer is filled ***************************************************)
	CASE State OF
	0:	
		IF Error
		THEN
			IF ResetTrig OR NOT Enable
			THEN
				Error										:= FALSE;
				ErrorId										:= 0;
				hr											:= S_OK;

				FileOpen(bExecute:=FALSE);	
				FileClose(bExecute:=FALSE);	
				FILEWRITE(bExecute:=FALSE);
			ELSIF NOT OPtions.0 AND hFile <> 0	
			THEN
				FileClose(bExecute:=TRUE , hFile := hFile);
				State										:= 3;
			END_IF
			
		ELSIF Enable
		THEN
			IF hr <> S_OK
			THEN //Method executed with error
				Error										:= TRUE;
				ErrorId										:= HRESULT_TO_ADSERROR(hr);
			ELSIF hFile = 0
			THEN
				WriteCounter								:= 0;	
				FileOpen(bExecute:= TRUE , sPathName:= CONCAT(Path,Filetype), nMode:=SEL(Options.7 ,FOPEN_MODEAPPEND,FOPEN_MODEWRITE) OR FOPEN_MODETEXT OR FOPEN_MODEPLUS );
				State										:= 1;		
			ELSIF ReadyToRead
			THEN
				FILEWRITE(bExecute:=TRUE ,hFile:= hFile , pWriteBuff := pDataToRead, cbWriteLen := SizeOfDataToRead);
				StartTimeWriteData							:= TIME();
				State										:= 2;			
			END_IF
		
		ELSIF hFile <> 0
		THEN //Not enabled
			IF NOT Empty
			THEN //Write rest of buffer		
				IF NOT ReadyToRead THEN setReadyToRead(TRUE); END_IF 
				FILEWRITE(bExecute:=ReadyToRead ,hFile:= hFile , pWriteBuff := pDataToRead, cbWriteLen := SizeOfDataToRead);
				StartTimeWriteData							:= TIME();
				State										:= 2;
			ELSE
				FileClose(bExecute:=TRUE , hFile := hFile);
				state										:= 3;	
			END_IF
        END_IF
     
	(* Open file *******************************************************************************)                                          	
	1:                       	
		FileOpen();                                     	
		IF NOT FileOpen.bBusy                           	
		THEN                                            	
			IF FileOpen.bError                          	
			THEN            
				Error										:= TRUE;                            	
				ErrorId										:= FileOpen.nErrId;
				State										:= 0;
			ELSE                                     	
				hFile										:= FileOpen.hFile;
				IF ReadyToRead
				THEN //Write request acitive
					FILEWRITE(bExecute:=TRUE ,hFile:= hFile , pWriteBuff := pDataToRead, cbWriteLen := SizeOfDataToRead);
					StartTimeWriteData						:= TIME();
					State									:= 2;
				ELSE
					State									:= 0;
				END_IF			
			END_IF
			FileOpen(bExecute:=FALSE);			
		END_IF

	(* Write data to file **********************************************************************)
	2: 
		FILEWRITE(hFile:= hFile);	
		IF NOT FILEWRITE.bBusy
		THEN
			IF FILEWRITE.bError
			THEN
				Error										:= TRUE;       
				ErrorId										:= FILEWRITE.nErrId;
				state										:= 0;
			ELSE                            
				WriteCounter								:= WriteCounter + 1;
				TimeWriteFile								:= TIME() - StartTimeWriteData;          	
				State										:= 3;	
				FileClose(bExecute:=TRUE , hFile := hFile);
			END_IF	
			setReadyToRead(FALSE); 
			FILEWRITE(bExecute:=FALSE);          		
		END_IF

	(* Close File ******************************************************************************)
	3: 
		FileClose(hFile := hFile);
		IF NOT FileClose.bBusy
		THEN
			IF FileClose.bError
			THEN
				Error										:= TRUE;       
				ErrorId										:= FileClose.nErrId;
				State										:= 0;
			ELSE                                        		
				hFile										:= 0;
				State										:= 0;
			END_IF
			FileClose(bExecute:=FALSE);
		END_IF
	ELSE
		;
	END_CASE

(* Ack ErrorIds **********************************************************)
	Busy 													:= State <> 0;
(**************************************************************************)

METHOD PUBLIC addData : HRESULT //Add data into write buffer and swap if if buffer is filled
VAR_INPUT
	pData													:	POINTER TO BYTE;
	SizeofData												:	UDINT;
END_VAR
IF NOT Error
THEN 
	IF SUPER^.addData(pData,SizeOfData) <> S_OK
	THEN
		ErrorId												:= HRESULT_TO_ADSERROR(hr);
		Error												:= TRUE;
	END_IF
ELSE
	addData													:= SEL(Error , E_HRESULTADSERR.INVALIDACCESS ,E_HRESULTADSERR.ERROR);
END_IF
END_METHOD

METHOD PUBLIC addString : HRESULT //Add string to write buffer and swap if buffer is filled
VAR_INPUT
	Data													:	T_MAXSTRING;
END_VAR
addString := This^.addData(ADR(Data),TO_UDINT(LEN(Data)));
END_METHOD

PROPERTY PUBLIC optKeepFileOnError : BOOL
GET
optKeepFileOnError := Options.0;
END_GET
SET
Options.0				:= optKeepFileOnError;
END_SET
END_PROPERTY

PROPERTY PUBLIC optStartNewFile : BOOL
GET
optStartNewFile := Options.7;
END_GET
SET
Options.7				:= optStartNewFile;
END_SET
END_PROPERTY

END_FUNCTION_BLOCK

// ---- TF11PlcSystem/ET_DoubleBuffer/DoubleBuffer.TcPOU
//Double buffer FB to fill one part of buffer while the other (filled) part can be read or processed meanwhile
//Variable "ReadyToRead" signals that recorded data can be read consistent by pointer "pDataToRead" 
//After the data are processed or copied, it is needed to call the method "setReadyToReady(Status := FALSE)" and release the buffer to be used if the other half is filled 
//With setReadyToReady(Status := TRUE) you can mark the current write buffer as "ReadyToRead" on demand and accessible via "pDataToRead"  (e.g. if no more data need to be recorded)
{attribute 'enable_dynamic_creation'}
FUNCTION_BLOCK DoubleBuffer
VAR_OUTPUT CONSTANT 	
END_VAR                     								
VAR_INPUT
	Overwrite												:	BOOL ; //Overwrite buffer read buffer if not released -> setReadyToRead(FALSE)        
	SizeOfMemory											: 	UDINT := 5120;	//Total size of dynamic allocated buffer (will be splited in half)	   								
END_VAR                     								
VAR_IN_OUT                  								
END_VAR                     								
VAR_OUTPUT       
	TimeFillBuffer											: 	TIME; //Last elapsed time to fill the buffer and set ReadyToRead=TRUE
	Full													:	BOOL; //Buffer is full
	Empty													:	BOOL := TRUE; //Buffer is empty 
	ReadyToRead												:	BOOL; //TRUE = Data are ready and can be read via "pDataToRead" to process 
	pDataToRead												:	POINTER TO BYTE; //Pointer to recorded data/filled buffer	
	SizeOfDataToRead										:	UDINT; //Count of bytes in filled buffer ready to ready 
{attribute 'displaymode':='hex'}
	hr														:	HRESULT; //Last result of method call
END_VAR                     								
VAR            
//local ************************************************************************************
	Interlock												:	BOOL; //Task interlock
	Buffer2Active											:	BOOL; //Indicates active buffer pointer 
	pBuffer1												: 	POINTER TO BYTE; //Pointer to start of allocated memory
	pBuffer2												: 	POINTER TO BYTE; //Pointer to second half of allocated memory
	StartTimeFillBuffer										:	TIME;
	
	MemSizeOfAllocatedMemory								: 	UDINT; //Total size of allocated memory
	MemSizeOfBuffer											: 	UDINT; //Size of split buffer
	MemSizeOfWriteBuffer									:	UDINT; //Actual size of recorded data


//trigger *********************************************************************************

//timer ***********************************************************************************

//instances ***********************************************************************************             								

//Dummys ****************************************************************************************

END_VAR

METHOD PUBLIC addData : HRESULT //Add data to write buffer and sets "ReadyToRead" if buffer is filled and data can be read to process 
VAR_INPUT
	pData													:	POINTER TO BYTE;
	SizeofData												:	UDINT;
END_VAR

IF pData <> 0 
THEN		
	//Allocate Memory to buffer messages
	IF pBuffer1 = 0
		OR SizeOfMemory > MemSizeOfAllocatedMemory 
	THEN //Allocate full memory with first entry 		
		IF NOT Allocate(SizeOfMemory)
		THEN
			addData := hr										:= E_HRESULTADSERR.NOMEMORY;
			RETURN;														
		END_IF					
	END_IF	

	IF MemSizeOfWriteBuffer = 0 THEN StartTimeFillBuffer := TIME(); END_IF
	
	//Change buffer if filled
	IF SizeofData + MemSizeOfWriteBuffer >= MemSizeOfBuffer
	THEN
		IF setReadyToRead(TRUE) <> S_OK
		THEN
			addData 											:= hr;
			RETURN;
		END_IF
	ELSE
		Full													:= FALSE;
		Empty													:= FALSE;
	END_IF
			
	//Copy data to buffer
	MEMCPY(SEL(Buffer2Active, pBuffer1, pBuffer2) + MemSizeOfWriteBuffer, pData, SizeofData);
	MemSizeOfWriteBuffer										:= MemSizeOfWriteBuffer + SizeofData;
	
	addData := hr												:= S_OK;
ELSE
	addData := hr												:= E_HRESULTADSERR.INVALIDPARM;
END_IF
END_METHOD

METHOD PUBLIC addString : HRESULT //Add string to write buffer and sets "ReadyToRead" if buffer is filled and data can be read to process 
VAR_INPUT
	Data													:	T_MAXSTRING;
END_VAR
addString := hr := addData(ADR(Data),TO_UDINT(LEN(Data)));
END_METHOD

METHOD PROTECTED FINAL allocate : BOOL //allocte buffer memory form router pool
VAR_INPUT
	SizeOfBuffer											:	UDINT;
END_VAR
VAR
	pDummy													:	POINTER TO BYTE;	
End_Var
IF SizeOfBuffer	= 0
THEN
	Allocate												:= FALSE;
	
ELSIF pBuffer1 = 0
THEN
	MemSizeOfAllocatedMemory								:= SizeOfBuffer;
	pBuffer1												:= __NEW(BYTE,MemSizeOfAllocatedMemory );
	MemSizeOfBuffer											:= MemSizeOfAllocatedMemory / 2;
	pBuffer2												:= pBuffer1 + MemSizeOfBuffer; 
	Buffer2Active											:= FALSE;
	MemSizeOfWriteBuffer									:= 0;
	
//	IF PARAM.ENABLE_DEBUG_MSG_DYNAMIC_MEM_ALLOCATION
//	THEN
//		AdsLogHint('EngineeringToolbox | FB DoubleBuffer | An instance allocated %s bytes from the dynamic memory of the ADS router memory pool', TO_STRING(MemSizeOfAllocatedMemory));
//	END_IF	
	Allocate												:= TRUE;
ELSIF SizeOfBuffer > MemSizeOfBuffer 
THEN //Since increased, allocate new memory
	
	pDummy													:= __NEW(BYTE, SizeOfBuffer); 

	IF SizeOfBuffer > MemSizeOfAllocatedMemory
	THEN //Size increased rescue data from old memory
		IF Buffer2Active
		THEN
			MEMCPY(pDummy,pBuffer2, MemSizeOfBuffer);
		ELSE
			MEMCPY(pDummy,pBuffer1, MemSizeOfBuffer);	
		END_IF
	END_IF

	__DELETE(pBuffer1);  //Delete reference to old memory
	
	MemSizeOfAllocatedMemory								:= SizeOfBuffer;
	pBuffer1												:= pDummy; //Take over new pointer to new memory
	Buffer2Active											:= FALSE;
	MemSizeOfBuffer											:= MemSizeOfAllocatedMemory / 2;
	pBuffer2												:= pBuffer1 + MemSizeOfBuffer; 
	MemSizeOfWriteBuffer										:= 0;
	
//	IF PARAM.ENABLE_DEBUG_MSG_DYNAMIC_MEM_ALLOCATION
//	THEN
//		AdsLogWarn('EngineeringToolbox | FB DoubleBuffer | Value of "SizeOfMemory" increased and an instance has an additional %s bytes allocated from the dynamic memory of the ADS router memory pool', TO_STRING(MemSizeOfAllocatedMemory));
//	END_IF
	
	Allocate												:= TRUE;
	
ELSE //Size decreased
	Allocate												:= TRUE;
END_IF
END_METHOD

METHOD PUBLIC copyData : HRESULT //Copy data from buffer (pDataToRead) into destination and reset "ReadyToReady" back to false if succeful executed 
VAR_INPUT
	pDest													:	POINTER TO BYTE; 
	SizeOfDest												:	UDINT; //Size of destination/data to copy
END_VAR
IF pDest <> 0 AND SizeOfDest > 0
	AND pDataToRead <> 0 
THEN
	MEMCPY(pDest, pDataToRead, MIN(SizeOfDest,SizeOfDataToRead));										
	hr		 												:= setReadyToRead(FALSE);	
	
ELSE
	IF pDataToRead = 0
	THEN
		hr													:= E_HRESULTADSERR.NOTREADY;
	ELSIF pDest = 0 
	THEN 
		hr													:= E_HRESULTADSERR.INVALIDPARM;
	ELSIF SizeOfDest = 0
	THEN
		hr													:= E_HRESULTADSERR.INVALIDPARM;	
	END_IF
END_IF
copyData													:= hr;
END_METHOD

METHOD FB_exit : BOOL
VAR_INPUT
	bInCopyCode : BOOL; // if TRUE, the exit method is called for exiting an instance that is copied afterwards (online change).
END_VAR
IF NOT bInCopyCode AND pBuffer1 <> 0
THEN //Release memory in case the PLC stopps
	__DELETE(pBuffer1);
END_IF
END_METHOD

{attribute 'monitoring' := 'call'}
PROPERTY PUBLIC fillLevel : INT //Buffer fill level 100% if both parts of buffer are filled
GET
IF MemSizeOfBuffer <> 0
THEN
	fillLevel												:= 	TO_INT((50.0 / TO_LREAL(MemSizeOfBuffer)) * TO_LREAL(MemSizeOfWriteBuffer))
																+ SEL(ReadyToRead, 0, TO_INT((50.0 / TO_LREAL(MemSizeOfBuffer)) * TO_LREAL(SizeOfDataToRead)));
ELSE
	fillLevel												:= 0;
END_IF
END_GET
END_PROPERTY

//Reset buffer 
METHOD PUBLIC reset : BOOL //TRUE if method is finnished
VAR_INPUT
END_VAR
TimeFillBuffer												:= T#0MS;
Full														:= FALSE; //Buffer is full
Empty														:= TRUE; //Buffer is empty 
ReadyToRead													:= FALSE;
SizeOfDataToRead											:= 0;
hr															:= S_OK;
MemSizeOfWriteBuffer										:= 0;
reset														:= TRUE;
END_METHOD

METHOD PUBLIC setReadyToRead : HRESULT //Status = FALSE to reset "ReadyToRead" and unlock buffer / Status = TRUE to mark current write buffer as filled and "ReadyToRead", accessible via "pDataToRead"
VAR_INPUT
	Status								:	BOOL; //FALSE to reset "ReadyToRead" or TRUE to set "ReadyToRead" and swap buffer 
END_VAR
IF TestAndSet(Interlock)
THEN
	IF NOT Status
	THEN
		ReadyToRead									:= FALSE;
		Full										:= FALSE;
		Empty										:= MemSizeOfWriteBuffer = 0;
		hr											:= S_OK;
	ELSIF Overwrite 
		OR NOT ReadyToRead
	THEN //Set ready to ready and swap buffer
		hr											:= SEL(swapBuffer(), E_HRESULTADSERR.ABORTED ,S_OK);
		TimeFillBuffer								:= TIME() - StartTimeFillBuffer;
		StartTimeFillBuffer							:= TIME();
		ReadyToRead									:= SizeOfDataToRead > 0;
		Full										:= FALSE;
		Empty										:= NOT ReadyToRead;
	ELSE
		TimeFillBuffer								:= TIME() - StartTimeFillBuffer;
		StartTimeFillBuffer							:= TIME();		
		Full										:= TRUE;
		Empty										:= FALSE;
		hr											:= E_HRESULTADSERR.ABORTED;	
	END_IF
		
	setReadyToRead									:= hr;
	Interlock										:= FALSE;
ELSE
	setReadyToRead									:= E_HRESULTADSERR.BUSY;
END_IF
END_METHOD

METHOD PROTECTED FINAL swapBuffer : BOOL //swap write and read buffer and asign filled buffer to pDataToRead
VAR_INPUT
END_VAR
pDataToRead													:= SEL(Buffer2Active, pBuffer1, pBuffer2);
SizeOfDataToRead											:= MemSizeOfWriteBuffer;	

Buffer2Active												:= NOT Buffer2Active;	

MemSizeOfWriteBuffer										:= 0;
swapBuffer													:= TRUE;
END_METHOD

END_FUNCTION_BLOCK

// ---- TF11PlcSystem/ET_DoubleBuffer/HRESULT_TO_ADSERROR.TcPOU
FUNCTION HRESULT_TO_ADSERROR     : E_AdsErr //Returns ADS error code from HRESULT (HRESULT HighWord offset = 16#9811, values <0 = Error, ==0 = OK, >0 = OK with Info   
VAR_INPUT
{attribute 'displaymode':='hex'}
	hr									:	HRESULT;
END_VAR
VAR
END_VAR

IF hr >= TO_DINT(16#98110000)
	AND hr <= TO_DINT(16#9811FFFF) 
THEN	
	HRESULT_TO_ADSERROR				:= TO_UDINT(hr - TO_DINT(16#98110000));
ELSE
	HRESULT_TO_ADSERROR				:= E_AdsErr.NOERR; //No ADS Error
END_IF

END_FUNCTION

// ---- TF11PlcSystem/File/FB_FileHandler.TcPOU
FUNCTION_BLOCK FB_FileHandler
VAR_INPUT
	sNetId: T_AmsNetId;
	sPathName: T_MaxString;
	
END_VAR
VAR_OUTPUT
END_VAR
VAR
	fbFileOpen : FB_FileOpen;
	fbFileClose : FB_FileClose;
	fbFileSeek : FB_FileSeek;
	fbFileTell : FB_FileTell;
	
	
	stepGetFileSize : INT;
	_hFile: UINT;
	
	
END_VAR

fbFileOpen(
	sNetId:= sNetId, 
	sPathName:= sPathName, 
	nMode:= FOPEN_MODEREAD OR FOPEN_MODEPLUS OR FOPEN_MODEBINARY, 
	ePath:= PATH_GENERIC, 
	bExecute:= , 
	tTimeout:= DEFAULT_ADS_TIMEOUT, 
	bBusy=> , 
	bError=> , 
	nErrId=> , 
	hFile=> _hFile);

METHOD GetFileSize : UDINT
VAR_INPUT
END_VAR
CASE stepGetFileSize OF
0:
	





END_CASE
END_METHOD

METHOD Open : BOOL
VAR_INPUT
END_VAR

fbFileOpen(bExecute := TRUE);
IF  NOT fbFileOpen.bBusy AND NOT fbFileOpen.bError THEN
	Open := TRUE;
END_IF
END_METHOD

END_FUNCTION_BLOCK

// ---- TF11PlcSystem/IO/DI_Button.TcPOU
{attribute 'no_check'}
(* 
按钮功能块 Button
按钮功能块，总体和Input差不多，针对按钮做了功能的完善可以将输入信号强制、反转或延迟
*)
FUNCTION_BLOCK DI_Button
VAR_INPUT
	Enable : BOOL := TRUE; (* 默认为True, False:不启用,除LED外输入无效  \ True:启用 *)
	Invert : BOOL := FALSE; (* False: 不反转Direct \ True: 在源头反转输入Invert Input *)
	Force : BOOL; (* 将输入强制为True, Force the In signal to True *)
	TrigOn : BOOL; (* 手动将Toggle模式输出置为True, 无论反转都是off优先 *)
	TrigOff : BOOL; (* 手动将Toggle模式输出置为False, 无论反转都是off优先 *)
	TrigOnDelay : BOOL; (* 手动将延迟后的Toggle模式输出置为True, 复位优先 *)
	TrigOffDelay : BOOL; (* 手动将延迟后的Toggle模式输出置为False, 复位优先 *)
	DelayTime : TIME := T#50MS; (* 延迟输出时间，T#0MS代表无延迟，也可充当滤波功能 *)
	LED AT%Q* : BOOL; (* 如果按钮有LED，绑定到LED的输出上，功能块内部本身不控制LED，需要外部程序通过该输入引脚控制 *)
END_VAR
VAR_OUTPUT
	Q : BOOL;(* 直接输出信号 *)
	Q_RT : BOOL;(* 输入信号的上升沿 *)
	Q_FT : BOOL;(* 输入信号的下降沿 *)
	Q_Tog : BOOL;(* Toggle模式输出，按一下切换为True，再按一下切换为False *)
	Q_Delay : BOOL;(* 经过延迟后的输出信号 *)
	Q_Delay_RT : BOOL;(* 经过延迟后的输出信号的上升沿 *)
	Q_Delay_FT : BOOL;(* 经过延迟后的输出信号的上升沿 *)
	Q_Delay_Tog : BOOL;(* 经过延迟后的Toggle模式输出，按一下切换为True，再按一下切换为False *)
	RawIn AT%I* :BOOL; (* 原始输入信号，未经强制、反转及延时 *) 
END_VAR
VAR
	rTrig, rTrig_Delay : R_TRIG;
	fTrig, fTrig_Delay : F_TRIG;
	tonDelay : TON;
END_VAR

